Yaskawa INFORM job: apremTRJ3.JBI

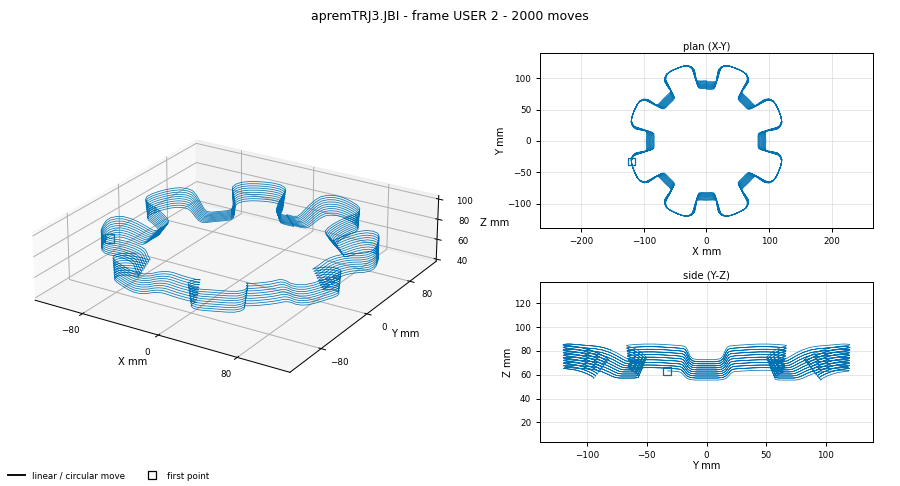
[picture p0: tool path of apremTRJ3.JBI in frame USER 2, 2000 of 2000 moves have a stored position in this frame; points joined in program order, loops and branches not executed]
/JOB
//NAME apremTRJ3
//POS
///NPOS 2000,0,0,0,0,0
///USER 2
///TOOL 1
///POSTYPE USER
///RECTAN
///RCONF 1,0,0,0,0,0,0,0,0,0,0,0,0,0,0,0,0,0,0,0,0,0,0,0
C00000=-119.725,-32.765,63.277,179.9256,-2.1058,0.0000
C00001=-118.418,-27.296,62.983,178.3163,-3.5512,0.0000
C00002=-115.167,-23.366,62.624,174.4376,-3.8430,0.0000
C00003=-110.519,-21.436,61.948,173.6854,-2.2369,0.0000
C00004=-105.464,-19.898,60.600,176.0753,-1.2711,0.0000
C00005=-100.994,-18.424,58.871,-179.3385,0.2539,0.0000
C00006=-97.711,-16.719,57.219,-170.3032,5.9788,0.0000
C00007=-95.932,-14.022,56.034,-167.2384,32.2356,0.0000
C00008=-95.724,-9.298,55.566,179.0443,38.8550,0.0000
C00009=-96.014,-4.602,55.545,177.5469,39.0995,0.0000
C00010=-96.126,0.000,55.559,-179.9998,39.1276,0.0000
C00011=-96.015,4.602,55.545,-177.5472,39.0996,0.0000
C00012=-95.724,9.298,55.566,-179.0464,38.8547,0.0000
C00013=-95.932,14.023,56.035,167.2390,32.2361,0.0000
C00014=-97.711,16.719,57.219,170.3032,5.9788,0.0000
C00015=-100.994,18.424,58.871,179.3385,0.2539,0.0000
C00016=-105.464,19.898,60.600,-176.0753,-1.2711,0.0000
C00017=-110.519,21.436,61.948,-173.6854,-2.2369,0.0000
C00018=-115.167,23.366,62.624,-174.4376,-3.8430,0.0000
C00019=-118.418,27.296,62.983,-178.3163,-3.5512,0.0000
C00020=-119.725,32.765,63.277,-179.9256,-2.1058,0.0000
C00021=-118.751,38.770,63.576,179.9642,-0.1157,0.0000
C00022=-116.678,44.821,63.773,179.9946,-0.0143,0.0000
C00023=-114.197,50.811,63.773,179.9937,-0.0139,0.0000
C00024=-111.384,56.555,63.576,179.9435,-0.1071,0.0000
C00025=-107.827,61.490,63.277,178.4580,-1.4368,0.0000
C00026=-103.035,64.433,62.983,176.3000,-1.3231,0.0000
C00027=-97.958,64.913,62.624,173.3627,1.2239,0.0000
C00028=-93.306,62.991,61.948,173.9567,2.8983,0.0000
C00029=-88.644,60.504,60.600,176.3265,1.8799,0.0000
C00030=-84.442,58.386,58.871,-179.3527,-0.2883,0.0000
C00031=-80.914,57.270,57.219,-168.9722,-2.6779,0.0000
C00032=-77.750,57.919,56.034,-148.7818,15.9473,0.0000
C00033=-74.261,61.112,55.566,-150.8450,30.1755,0.0000
C00034=-71.147,64.638,55.545,-151.4385,31.1712,0.0000
C00035=-67.972,67.972,55.559,-150.0917,29.9081,0.0000
C00036=-64.639,71.146,55.545,-148.8289,28.5617,0.0000
C00037=-61.112,74.261,55.566,-149.8258,29.1559,0.0000
C00038=-57.919,77.750,56.035,-164.0518,31.2182,0.0000
C00039=-57.270,80.914,57.219,177.3221,11.0278,0.0000
C00040=-58.386,84.442,58.871,179.7117,0.6473,0.0000
C00041=-60.504,88.644,60.600,-178.1201,-3.6735,0.0000
C00042=-62.991,93.306,61.948,-177.1017,-6.0433,0.0000
C00043=-64.913,97.958,62.624,-178.7761,-6.6373,0.0000
C00044=-64.433,103.035,62.983,178.6769,-3.7000,0.0000
C00045=-61.490,107.827,63.277,178.5632,-1.5420,0.0000
C00046=-56.555,111.384,63.576,179.8929,-0.0565,0.0000
C00047=-50.811,114.197,63.773,179.9861,-0.0063,0.0000
C00048=-44.821,116.678,63.773,179.9857,-0.0054,0.0000
C00049=-38.770,118.751,63.576,179.8843,-0.0358,0.0000
C00050=-32.765,119.725,63.277,177.8942,0.0744,0.0000
C00051=-27.296,118.418,62.983,176.4488,1.6837,0.0000
C00052=-23.366,115.167,62.624,176.1570,5.5624,0.0000
C00053=-21.436,110.519,61.948,177.7631,6.3146,0.0000
C00054=-19.898,105.464,60.600,178.7289,3.9247,0.0000
C00055=-18.424,100.994,58.871,-179.7461,-0.6615,0.0000
C00056=-16.719,97.711,57.219,-174.0212,-9.6968,0.0000
C00057=-14.023,95.932,56.035,-147.7639,-12.7610,0.0000
C00058=-9.298,95.724,55.566,-141.1453,0.9536,0.0000
C00059=-4.602,96.015,55.545,-140.9004,2.4528,0.0000
C00060=0.000,96.126,55.559,-140.8724,0.0002,0.0000
C00061=0.000,94.736,57.264,-140.7733,0.0001,0.0000
C00062=4.475,94.629,57.250,-140.8009,-2.4427,0.0000
C00063=9.084,94.351,57.271,-141.0650,-0.7004,0.0000
C00064=13.760,94.602,57.767,-148.3519,13.4830,0.0000
C00065=16.395,96.491,59.021,-174.9739,8.8071,0.0000
C00066=18.049,99.951,60.772,-179.9988,0.0034,0.0000
C00067=19.486,104.658,62.604,178.6708,-4.3590,0.0000
C00068=20.989,109.986,64.035,177.7869,-6.6807,0.0000
C00069=22.877,114.901,64.752,176.1277,-5.9675,0.0000
C00070=26.834,118.363,65.133,176.2739,-1.8689,0.0000
C00071=32.398,119.792,65.445,177.8036,-0.1013,0.0000
C00072=38.538,118.828,65.762,179.8764,0.0380,0.0000
C00073=44.742,116.708,65.972,179.9849,0.0057,0.0000
C00074=50.888,114.162,65.972,179.9853,0.0067,0.0000
C00075=56.774,111.274,65.762,179.8857,0.0605,0.0000
C00076=61.797,107.615,65.445,178.5181,1.6250,0.0000
C00077=64.721,102.670,65.133,178.6837,3.9541,0.0000
C00078=65.071,97.424,64.752,-178.5077,6.9431,0.0000
C00079=62.931,92.614,64.035,-176.8235,6.2858,0.0000
C00080=60.226,87.783,62.604,-177.8528,4.0217,0.0000
C00081=57.914,83.439,60.772,179.9985,-0.0033,0.0000
C00082=56.637,79.823,59.021,177.2881,-9.7451,0.0000
C00083=57.164,76.624,57.767,-165.0885,-31.1896,0.0000
C00084=60.292,73.139,57.271,-149.8896,-29.3635,0.0000
C00085=63.749,70.077,57.250,-148.7486,-28.6574,0.0000
C00086=66.989,66.989,57.264,-150.0043,-29.9958,0.0000
C00087=70.077,63.749,57.250,-151.3424,-31.2513,0.0000
C00088=73.140,60.292,57.271,-150.6355,-30.1090,0.0000
C00089=76.624,57.164,57.767,-148.8104,-14.9124,0.0000
C00090=79.823,56.637,59.021,-170.2549,2.7119,0.0000
C00091=83.439,57.914,60.772,-179.9967,0.0015,0.0000
C00092=87.783,60.226,62.604,175.9783,-2.1472,0.0000
C00093=92.614,62.931,64.035,173.7142,-3.1765,0.0000
C00094=97.424,65.071,64.752,173.0569,-1.4923,0.0000
C00095=102.670,64.721,65.133,176.0459,1.3163,0.0000
C00096=107.615,61.797,65.445,178.3750,1.4819,0.0000
C00097=111.274,56.774,65.762,179.9395,0.1143,0.0000
C00098=114.162,50.888,65.972,179.9933,0.0147,0.0000
C00099=116.708,44.742,65.972,179.9943,0.0151,0.0000
C00100=118.828,38.538,65.762,179.9620,0.1236,0.0000
C00101=119.792,32.398,65.445,-179.8987,2.1964,0.0000
C00102=118.363,26.834,65.133,-178.1311,3.7261,0.0000
C00103=114.901,22.877,64.752,-174.0325,3.8723,0.0000
C00104=109.986,20.989,64.035,-173.3193,2.2131,0.0000
C00105=104.658,19.486,62.604,-175.6410,1.3292,0.0000
C00106=99.951,18.049,60.772,179.9966,-0.0012,0.0000
C00107=96.491,16.395,59.021,171.1929,-5.0261,0.0000
C00108=94.602,13.760,57.767,166.5170,-31.6481,0.0000
C00109=94.351,9.084,57.271,-179.2996,-38.9350,0.0000
C00110=94.629,4.475,57.250,-177.5573,-39.1991,0.0000
C00111=94.736,0.000,57.264,179.9999,-39.2267,0.0000
C00112=94.629,-4.475,57.250,177.5575,-39.1991,0.0000
C00113=94.351,-9.084,57.271,179.3018,-38.9347,0.0000
C00114=94.602,-13.760,57.767,-166.5176,-31.6486,0.0000
C00115=96.491,-16.395,59.021,-171.1929,-5.0261,0.0000
C00116=99.951,-18.049,60.772,-179.9966,-0.0012,0.0000
C00117=104.658,-19.486,62.604,175.6410,1.3292,0.0000
C00118=109.986,-20.989,64.035,173.3193,2.2131,0.0000
C00119=114.901,-22.877,64.752,174.0325,3.8723,0.0000
C00120=118.363,-26.834,65.133,178.1311,3.7261,0.0000
C00121=119.792,-32.398,65.445,179.8987,2.1964,0.0000
C00122=118.828,-38.538,65.762,-179.9620,0.1236,0.0000
C00123=116.708,-44.742,65.972,-179.9943,0.0151,0.0000
C00124=114.162,-50.888,65.972,-179.9933,0.0147,0.0000
C00125=111.274,-56.774,65.762,-179.9395,0.1143,0.0000
C00126=107.615,-61.797,65.445,-178.3750,1.4819,0.0000
C00127=102.670,-64.721,65.133,-176.0459,1.3163,0.0000
C00128=97.424,-65.071,64.752,-173.0569,-1.4923,0.0000
C00129=92.614,-62.931,64.035,-173.7142,-3.1765,0.0000
C00130=87.783,-60.226,62.604,-175.9783,-2.1472,0.0000
C00131=83.439,-57.914,60.772,179.9967,0.0015,0.0000
C00132=79.823,-56.637,59.021,170.2549,2.7119,0.0000
C00133=76.624,-57.164,57.767,148.8104,-14.9115,0.0000
C00134=73.139,-60.292,57.271,150.6365,-30.1104,0.0000
C00135=70.077,-63.749,57.250,151.3426,-31.2514,0.0000
C00136=66.989,-66.989,57.264,150.0042,-29.9957,0.0000
C00137=63.749,-70.077,57.250,148.7487,-28.6576,0.0000
C00138=60.292,-73.140,57.271,149.8910,-29.3645,0.0000
C00139=57.164,-76.624,57.767,165.0876,-31.1896,0.0000
C00140=56.637,-79.823,59.021,-177.2881,-9.7451,0.0000
C00141=57.914,-83.439,60.772,-179.9985,-0.0033,0.0000
C00142=60.226,-87.783,62.604,177.8528,4.0217,0.0000
C00143=62.931,-92.614,64.035,176.8235,6.2858,0.0000
C00144=65.071,-97.424,64.752,178.5077,6.9431,0.0000
C00145=64.721,-102.670,65.133,-178.6837,3.9541,0.0000
C00146=61.797,-107.615,65.445,-178.5181,1.6250,0.0000
C00147=56.774,-111.274,65.762,-179.8857,0.0605,0.0000
C00148=50.888,-114.162,65.972,-179.9853,0.0067,0.0000
C00149=44.742,-116.708,65.972,-179.9849,0.0057,0.0000
C00150=38.538,-118.828,65.762,-179.8764,0.0380,0.0000
C00151=32.398,-119.792,65.445,-177.8036,-0.1013,0.0000
C00152=26.834,-118.363,65.133,-176.2739,-1.8689,0.0000
C00153=22.877,-114.901,64.752,-176.1277,-5.9675,0.0000
C00154=20.989,-109.986,64.035,-177.7869,-6.6807,0.0000
C00155=19.486,-104.658,62.604,-178.6708,-4.3590,0.0000
C00156=18.049,-99.951,60.772,179.9988,0.0034,0.0000
C00157=16.395,-96.491,59.021,174.9739,8.8071,0.0000
C00158=13.760,-94.602,57.767,148.3519,13.4830,0.0000
C00159=9.084,-94.351,57.271,141.0650,-0.7004,0.0000
C00160=4.475,-94.629,57.250,140.8009,-2.4427,0.0000
C00161=0.000,-94.736,57.264,140.7733,0.0001,0.0000
C00162=0.000,-94.736,57.264,140.7733,0.0001,0.0000
C00163=-4.475,-94.629,57.250,140.8009,2.4425,0.0000
C00164=-9.084,-94.351,57.271,141.0653,0.6982,0.0000
C00165=-13.760,-94.602,57.767,148.3514,-13.4824,0.0000
C00166=-16.395,-96.491,59.021,174.9739,-8.8071,0.0000
C00167=-18.049,-99.951,60.772,179.9988,-0.0034,0.0000
C00168=-19.486,-104.658,62.604,-178.6708,4.3590,0.0000
C00169=-20.989,-109.986,64.035,-177.7869,6.6807,0.0000
C00170=-22.877,-114.901,64.752,-176.1277,5.9675,0.0000
C00171=-26.834,-118.363,65.133,-176.2739,1.8689,0.0000
C00172=-32.398,-119.792,65.445,-177.8036,0.1013,0.0000
C00173=-38.538,-118.828,65.762,-179.8764,-0.0380,0.0000
C00174=-44.742,-116.708,65.972,-179.9849,-0.0057,0.0000
C00175=-50.888,-114.162,65.972,-179.9853,-0.0067,0.0000
C00176=-56.774,-111.274,65.762,-179.8857,-0.0605,0.0000
C00177=-61.797,-107.615,65.445,-178.5181,-1.6250,0.0000
C00178=-64.721,-102.670,65.133,-178.6837,-3.9541,0.0000
C00179=-65.071,-97.424,64.752,178.5077,-6.9431,0.0000
C00180=-62.931,-92.614,64.035,176.8235,-6.2858,0.0000
C00181=-60.226,-87.783,62.604,177.8528,-4.0217,0.0000
C00182=-57.914,-83.439,60.772,-179.9985,0.0033,0.0000
C00183=-56.637,-79.823,59.021,-177.2881,9.7451,0.0000
C00184=-57.164,-76.624,57.767,165.0885,31.1896,0.0000
C00185=-60.292,-73.139,57.271,149.8896,29.3635,0.0000
C00186=-63.749,-70.077,57.250,148.7486,28.6574,0.0000
C00187=-66.989,-66.989,57.264,150.0043,29.9958,0.0000
C00188=-70.077,-63.749,57.250,151.3424,31.2513,0.0000
C00189=-73.140,-60.292,57.271,150.6355,30.1090,0.0000
C00190=-76.624,-57.164,57.767,148.8104,14.9124,0.0000
C00191=-79.823,-56.637,59.021,170.2549,-2.7119,0.0000
C00192=-83.439,-57.914,60.772,179.9967,-0.0015,0.0000
C00193=-87.783,-60.226,62.604,-175.9783,2.1472,0.0000
C00194=-92.614,-62.931,64.035,-173.7142,3.1765,0.0000
C00195=-97.424,-65.071,64.752,-173.0569,1.4923,0.0000
C00196=-102.670,-64.721,65.133,-176.0459,-1.3163,0.0000
C00197=-107.615,-61.797,65.445,-178.3750,-1.4819,0.0000
C00198=-111.274,-56.774,65.762,-179.9395,-0.1143,0.0000
C00199=-114.162,-50.888,65.972,-179.9933,-0.0147,0.0000
C00200=-116.708,-44.742,65.972,-179.9943,-0.0151,0.0000
C00201=-118.828,-38.538,65.762,-179.9620,-0.1236,0.0000
C00202=-119.792,-32.398,65.445,179.8987,-2.1964,0.0000
C00203=-118.363,-26.834,65.133,178.1311,-3.7261,0.0000
C00204=-114.901,-22.877,64.752,174.0325,-3.8723,0.0000
C00205=-109.986,-20.989,64.035,173.3193,-2.2131,0.0000
C00206=-104.658,-19.486,62.604,175.6410,-1.3292,0.0000
C00207=-99.951,-18.049,60.772,-179.9966,0.0012,0.0000
C00208=-96.491,-16.395,59.021,-171.1929,5.0261,0.0000
C00209=-94.602,-13.760,57.767,-166.5170,31.6481,0.0000
C00210=-94.351,-9.084,57.271,179.2996,38.9350,0.0000
C00211=-94.629,-4.475,57.250,177.5573,39.1991,0.0000
C00212=-94.736,0.000,57.264,-179.9999,39.2267,0.0000
C00213=-94.629,4.475,57.250,-177.5575,39.1991,0.0000
C00214=-94.351,9.084,57.271,-179.3018,38.9347,0.0000
C00215=-94.602,13.760,57.767,166.5176,31.6486,0.0000
C00216=-96.491,16.395,59.021,171.1929,5.0261,0.0000
C00217=-99.951,18.049,60.772,179.9966,0.0012,0.0000
C00218=-104.658,19.486,62.604,-175.6410,-1.3292,0.0000
C00219=-109.986,20.989,64.035,-173.3193,-2.2131,0.0000
C00220=-114.901,22.877,64.752,-174.0325,-3.8723,0.0000
C00221=-118.363,26.834,65.133,-178.1311,-3.7261,0.0000
C00222=-119.792,32.398,65.445,-179.8987,-2.1964,0.0000
C00223=-118.828,38.538,65.762,179.9620,-0.1236,0.0000
C00224=-116.708,44.742,65.972,179.9943,-0.0151,0.0000
C00225=-114.162,50.888,65.972,179.9933,-0.0147,0.0000
C00226=-111.274,56.774,65.762,179.9395,-0.1143,0.0000
C00227=-107.615,61.797,65.445,178.3750,-1.4819,0.0000
C00228=-102.670,64.721,65.133,176.0459,-1.3163,0.0000
C00229=-97.424,65.071,64.752,173.0569,1.4923,0.0000
C00230=-92.614,62.931,64.035,173.7142,3.1765,0.0000
C00231=-87.783,60.226,62.604,175.9783,2.1472,0.0000
C00232=-83.439,57.914,60.772,-179.9967,-0.0015,0.0000
C00233=-79.823,56.637,59.021,-170.2549,-2.7119,0.0000
C00234=-76.624,57.164,57.767,-148.8104,14.9115,0.0000
C00235=-73.139,60.292,57.271,-150.6365,30.1104,0.0000
C00236=-70.077,63.749,57.250,-151.3426,31.2514,0.0000
C00237=-66.989,66.989,57.264,-150.0042,29.9957,0.0000
C00238=-63.749,70.077,57.250,-148.7487,28.6576,0.0000
C00239=-60.292,73.140,57.271,-149.8910,29.3645,0.0000
C00240=-57.164,76.624,57.767,-165.0876,31.1896,0.0000
C00241=-56.637,79.823,59.021,177.2881,9.7451,0.0000
C00242=-57.914,83.439,60.772,179.9985,0.0033,0.0000
C00243=-60.226,87.783,62.604,-177.8528,-4.0217,0.0000
C00244=-62.931,92.614,64.035,-176.8235,-6.2858,0.0000
C00245=-65.071,97.424,64.752,-178.5077,-6.9431,0.0000
C00246=-64.721,102.670,65.133,178.6837,-3.9541,0.0000
C00247=-61.797,107.615,65.445,178.5181,-1.6250,0.0000
C00248=-56.774,111.274,65.762,179.8857,-0.0605,0.0000
C00249=-50.888,114.162,65.972,179.9853,-0.0067,0.0000
C00250=-44.742,116.708,65.972,179.9849,-0.0057,0.0000
C00251=-38.538,118.828,65.762,179.8764,-0.0380,0.0000
C00252=-32.398,119.792,65.445,177.8036,0.1013,0.0000
C00253=-26.834,118.363,65.133,176.2739,1.8689,0.0000
C00254=-22.877,114.901,64.752,176.1277,5.9675,0.0000
C00255=-20.989,109.986,64.035,177.7869,6.6807,0.0000
C00256=-19.486,104.658,62.604,178.6708,4.3590,0.0000
C00257=-18.049,99.951,60.772,-179.9988,-0.0034,0.0000
C00258=-16.395,96.491,59.021,-174.9739,-8.8071,0.0000
C00259=-13.760,94.602,57.767,-148.3514,-13.4824,0.0000
C00260=-9.084,94.351,57.271,-141.0653,0.6982,0.0000
C00261=-4.475,94.629,57.250,-140.8009,2.4425,0.0000
C00262=0.000,94.736,57.264,-140.7733,0.0001,0.0000
C00263=0.000,93.344,58.968,-140.7215,0.0000,0.0000
C00264=4.348,93.242,58.953,-140.7485,-2.4271,0.0000
C00265=8.870,92.975,58.975,-141.0344,-0.4357,0.0000
C00266=13.498,93.270,59.499,-149.0201,14.1329,0.0000
C00267=16.071,95.271,60.823,-175.8165,7.9019,0.0000
C00268=17.674,98.909,62.673,179.7950,-0.6064,0.0000
C00269=19.074,103.853,64.610,178.6348,-4.7423,0.0000
C00270=20.544,109.456,66.124,177.8284,-6.9903,0.0000
C00271=22.391,114.637,66.882,176.1347,-6.3202,0.0000
C00272=26.375,118.308,67.284,176.1293,-2.0440,0.0000
C00273=32.034,119.858,67.614,177.7255,-0.1282,0.0000
C00274=38.307,118.904,67.949,179.8694,0.0400,0.0000
C00275=44.664,116.738,68.170,179.9841,0.0060,0.0000
C00276=50.965,114.128,68.170,179.9845,0.0070,0.0000
C00277=56.991,111.165,67.949,179.8794,0.0641,0.0000
C00278=62.101,107.404,67.614,178.4818,1.6994,0.0000
C00279=65.006,102.306,67.284,178.7050,4.1797,0.0000
C00280=65.228,96.893,66.882,-178.2506,7.1867,0.0000
C00281=62.871,91.924,66.124,-176.5728,6.4761,0.0000
C00282=59.948,86.923,64.610,-177.6059,4.3183,0.0000
C00283=57.442,82.437,62.673,-179.7162,0.5738,0.0000
C00284=56.002,78.731,60.823,177.3422,-8.5232,0.0000
C00285=56.408,75.496,59.499,-166.1532,-31.0723,0.0000
C00286=59.471,72.016,58.975,-150.0031,-29.5326,0.0000
C00287=62.858,69.007,58.953,-148.7116,-28.7135,0.0000
C00288=66.004,66.004,58.968,-149.9585,-30.0416,0.0000
C00289=69.006,62.858,58.953,-151.2864,-31.2884,0.0000
C00290=72.016,59.471,58.975,-150.4665,-29.9954,0.0000
C00291=75.496,56.408,59.499,-148.9276,-13.8477,0.0000
C00292=78.731,56.002,60.823,-171.4768,2.6578,0.0000
C00293=82.437,57.442,62.673,179.4262,-0.2838,0.0000
C00294=86.923,59.948,64.610,175.6817,-2.3941,0.0000
C00295=91.924,62.871,66.124,173.5239,-3.4272,0.0000
C00296=96.893,65.228,66.882,172.8133,-1.7494,0.0000
C00297=102.306,65.006,67.284,175.8203,1.2950,0.0000
C00298=107.404,62.101,67.614,178.3006,1.5182,0.0000
C00299=111.165,56.991,67.949,179.9359,0.1206,0.0000
C00300=114.128,50.965,68.170,179.9930,0.0155,0.0000
C00301=116.738,44.664,68.170,179.9940,0.0159,0.0000
C00302=118.904,38.307,67.949,179.9600,0.1306,0.0000
C00303=119.858,32.034,67.614,-179.8718,2.2745,0.0000
C00304=118.308,26.375,67.284,-177.9560,3.8707,0.0000
C00305=114.637,22.391,66.882,-173.6798,3.8653,0.0000
C00306=109.456,20.544,66.124,-173.0097,2.1716,0.0000
C00307=103.853,19.074,64.610,-175.2577,1.3652,0.0000
C00308=98.909,17.674,62.673,-179.3936,0.2050,0.0000
C00309=95.271,16.071,60.823,172.0981,-4.1835,0.0000
C00310=93.270,13.498,59.499,165.8671,-30.9799,0.0000
C00311=92.975,8.870,58.975,-179.5643,-38.9656,0.0000
C00312=93.242,4.348,58.953,-177.5729,-39.2515,0.0000
C00313=93.344,0.000,58.968,180.0000,-39.2785,0.0000
C00314=93.242,-4.348,58.953,177.5731,-39.2515,0.0000
C00315=92.976,-8.870,58.975,179.5666,-38.9653,0.0000
C00316=93.271,-13.498,59.499,-165.8676,-30.9804,0.0000
C00317=95.271,-16.071,60.823,-172.0981,-4.1835,0.0000
C00318=98.909,-17.674,62.673,179.3936,0.2050,0.0000
C00319=103.853,-19.074,64.610,175.2577,1.3652,0.0000
C00320=109.456,-20.544,66.124,173.0097,2.1716,0.0000
C00321=114.637,-22.391,66.882,173.6798,3.8653,0.0000
C00322=118.308,-26.375,67.284,177.9560,3.8707,0.0000
C00323=119.858,-32.034,67.614,179.8718,2.2745,0.0000
C00324=118.904,-38.307,67.949,-179.9600,0.1306,0.0000
C00325=116.738,-44.664,68.170,-179.9940,0.0159,0.0000
C00326=114.128,-50.965,68.170,-179.9930,0.0155,0.0000
C00327=111.165,-56.991,67.949,-179.9359,0.1206,0.0000
C00328=107.404,-62.101,67.614,-178.3006,1.5182,0.0000
C00329=102.306,-65.006,67.284,-175.8203,1.2950,0.0000
C00330=96.893,-65.228,66.882,-172.8133,-1.7494,0.0000
C00331=91.924,-62.871,66.124,-173.5239,-3.4272,0.0000
C00332=86.923,-59.948,64.610,-175.6817,-2.3941,0.0000
C00333=82.437,-57.442,62.673,-179.4262,-0.2838,0.0000
C00334=78.731,-56.002,60.823,171.4768,2.6578,0.0000
C00335=75.496,-56.408,59.499,148.9277,-13.8468,0.0000
C00336=72.016,-59.471,58.975,150.4674,-29.9969,0.0000
C00337=69.007,-62.858,58.953,151.2865,-31.2884,0.0000
C00338=66.004,-66.004,58.968,149.9584,-30.0415,0.0000
C00339=62.858,-69.006,58.953,148.7116,-28.7136,0.0000
C00340=59.471,-72.016,58.975,150.0046,-29.5335,0.0000
C00341=56.408,-75.496,59.499,166.1523,-31.0724,0.0000
C00342=56.002,-78.731,60.823,-177.3422,-8.5232,0.0000
C00343=57.442,-82.437,62.673,179.7162,0.5738,0.0000
C00344=59.948,-86.923,64.610,177.6059,4.3183,0.0000
C00345=62.871,-91.924,66.124,176.5728,6.4761,0.0000
C00346=65.228,-96.893,66.882,178.2506,7.1867,0.0000
C00347=65.006,-102.306,67.284,-178.7050,4.1797,0.0000
C00348=62.101,-107.404,67.614,-178.4818,1.6994,0.0000
C00349=56.991,-111.165,67.949,-179.8794,0.0641,0.0000
C00350=50.965,-114.128,68.170,-179.9845,0.0070,0.0000
C00351=44.664,-116.738,68.170,-179.9841,0.0060,0.0000
C00352=38.307,-118.904,67.949,-179.8694,0.0400,0.0000
C00353=32.034,-119.858,67.614,-177.7255,-0.1282,0.0000
C00354=26.375,-118.308,67.284,-176.1293,-2.0440,0.0000
C00355=22.391,-114.637,66.882,-176.1347,-6.3202,0.0000
C00356=20.544,-109.456,66.124,-177.8284,-6.9903,0.0000
C00357=19.074,-103.853,64.610,-178.6348,-4.7423,0.0000
C00358=17.674,-98.909,62.673,-179.7950,-0.6064,0.0000
C00359=16.071,-95.271,60.823,175.8165,7.9019,0.0000
C00360=13.498,-93.270,59.499,149.0201,14.1329,0.0000
C00361=8.870,-92.975,58.975,141.0344,-0.4357,0.0000
C00362=4.348,-93.242,58.953,140.7485,-2.4271,0.0000
C00363=0.000,-93.344,58.968,140.7215,0.0000,0.0000
C00364=0.000,-93.344,58.968,140.7215,0.0000,0.0000
C00365=-4.348,-93.242,58.953,140.7485,2.4269,0.0000
C00366=-8.870,-92.976,58.975,141.0347,0.4334,0.0000
C00367=-13.498,-93.271,59.499,149.0196,-14.1324,0.0000
C00368=-16.071,-95.271,60.823,175.8165,-7.9019,0.0000
C00369=-17.674,-98.909,62.673,-179.7950,0.6064,0.0000
C00370=-19.074,-103.853,64.610,-178.6348,4.7423,0.0000
C00371=-20.544,-109.456,66.124,-177.8284,6.9903,0.0000
C00372=-22.391,-114.637,66.882,-176.1347,6.3202,0.0000
C00373=-26.375,-118.308,67.284,-176.1293,2.0440,0.0000
C00374=-32.034,-119.858,67.614,-177.7255,0.1282,0.0000
C00375=-38.307,-118.904,67.949,-179.8694,-0.0400,0.0000
C00376=-44.664,-116.738,68.170,-179.9841,-0.0060,0.0000
C00377=-50.965,-114.128,68.170,-179.9845,-0.0070,0.0000
C00378=-56.991,-111.165,67.949,-179.8794,-0.0641,0.0000
C00379=-62.101,-107.404,67.614,-178.4818,-1.6994,0.0000
C00380=-65.006,-102.306,67.284,-178.7050,-4.1797,0.0000
C00381=-65.228,-96.893,66.882,178.2506,-7.1867,0.0000
C00382=-62.871,-91.924,66.124,176.5728,-6.4761,0.0000
C00383=-59.948,-86.923,64.610,177.6059,-4.3183,0.0000
C00384=-57.442,-82.437,62.673,179.7162,-0.5738,0.0000
C00385=-56.002,-78.731,60.823,-177.3422,8.5232,0.0000
C00386=-56.408,-75.496,59.499,166.1532,31.0723,0.0000
C00387=-59.471,-72.016,58.975,150.0031,29.5326,0.0000
C00388=-62.858,-69.007,58.953,148.7116,28.7135,0.0000
C00389=-66.004,-66.004,58.968,149.9585,30.0416,0.0000
C00390=-69.006,-62.858,58.953,151.2864,31.2884,0.0000
C00391=-72.016,-59.471,58.975,150.4665,29.9954,0.0000
C00392=-75.496,-56.408,59.499,148.9276,13.8477,0.0000
C00393=-78.731,-56.002,60.823,171.4768,-2.6578,0.0000
C00394=-82.437,-57.442,62.673,-179.4262,0.2838,0.0000
C00395=-86.923,-59.948,64.610,-175.6817,2.3941,0.0000
C00396=-91.924,-62.871,66.124,-173.5239,3.4272,0.0000
C00397=-96.893,-65.228,66.882,-172.8133,1.7494,0.0000
C00398=-102.306,-65.006,67.284,-175.8203,-1.2950,0.0000
C00399=-107.404,-62.101,67.614,-178.3006,-1.5182,0.0000
C00400=-111.165,-56.991,67.949,-179.9359,-0.1206,0.0000
C00401=-114.128,-50.965,68.170,-179.9930,-0.0155,0.0000
C00402=-116.738,-44.664,68.170,-179.9940,-0.0159,0.0000
C00403=-118.904,-38.307,67.949,-179.9600,-0.1306,0.0000
C00404=-119.858,-32.034,67.614,179.8718,-2.2745,0.0000
C00405=-118.308,-26.375,67.284,177.9560,-3.8707,0.0000
C00406=-114.637,-22.391,66.882,173.6798,-3.8653,0.0000
C00407=-109.456,-20.544,66.124,173.0097,-2.1716,0.0000
C00408=-103.853,-19.074,64.610,175.2577,-1.3652,0.0000
C00409=-98.909,-17.674,62.673,179.3936,-0.2050,0.0000
C00410=-95.271,-16.071,60.823,-172.0981,4.1835,0.0000
C00411=-93.270,-13.498,59.499,-165.8671,30.9799,0.0000
C00412=-92.975,-8.870,58.975,179.5643,38.9656,0.0000
C00413=-93.242,-4.348,58.953,177.5729,39.2515,0.0000
C00414=-93.344,0.000,58.968,-180.0000,39.2785,0.0000
C00415=-93.242,4.348,58.953,-177.5731,39.2515,0.0000
C00416=-92.976,8.870,58.975,-179.5666,38.9653,0.0000
C00417=-93.271,13.498,59.499,165.8676,30.9804,0.0000
C00418=-95.271,16.071,60.823,172.0981,4.1835,0.0000
C00419=-98.909,17.674,62.673,-179.3936,-0.2050,0.0000
C00420=-103.853,19.074,64.610,-175.2577,-1.3652,0.0000
C00421=-109.456,20.544,66.124,-173.0097,-2.1716,0.0000
C00422=-114.637,22.391,66.882,-173.6798,-3.8653,0.0000
C00423=-118.308,26.375,67.284,-177.9560,-3.8707,0.0000
C00424=-119.858,32.034,67.614,-179.8718,-2.2745,0.0000
C00425=-118.904,38.307,67.949,179.9600,-0.1306,0.0000
C00426=-116.738,44.664,68.170,179.9940,-0.0159,0.0000
C00427=-114.128,50.965,68.170,179.9930,-0.0155,0.0000
C00428=-111.165,56.991,67.949,179.9359,-0.1206,0.0000
C00429=-107.404,62.101,67.614,178.3006,-1.5182,0.0000
C00430=-102.306,65.006,67.284,175.8203,-1.2950,0.0000
C00431=-96.893,65.228,66.882,172.8133,1.7494,0.0000
C00432=-91.924,62.871,66.124,173.5239,3.4272,0.0000
C00433=-86.923,59.948,64.610,175.6817,2.3941,0.0000
C00434=-82.437,57.442,62.673,179.4262,0.2838,0.0000
C00435=-78.731,56.002,60.823,-171.4768,-2.6578,0.0000
C00436=-75.496,56.408,59.499,-148.9277,13.8468,0.0000
C00437=-72.016,59.471,58.975,-150.4674,29.9969,0.0000
C00438=-69.007,62.858,58.953,-151.2865,31.2884,0.0000
C00439=-66.004,66.004,58.968,-149.9584,30.0415,0.0000
C00440=-62.858,69.006,58.953,-148.7116,28.7136,0.0000
C00441=-59.471,72.016,58.975,-150.0046,29.5335,0.0000
C00442=-56.408,75.496,59.499,-166.1523,31.0724,0.0000
C00443=-56.002,78.731,60.823,177.3422,8.5232,0.0000
C00444=-57.442,82.437,62.673,-179.7162,-0.5738,0.0000
C00445=-59.948,86.923,64.610,-177.6059,-4.3183,0.0000
C00446=-62.871,91.924,66.124,-176.5728,-6.4761,0.0000
C00447=-65.228,96.893,66.882,-178.2506,-7.1867,0.0000
C00448=-65.006,102.306,67.284,178.7050,-4.1797,0.0000
C00449=-62.101,107.404,67.614,178.4818,-1.6994,0.0000
C00450=-56.991,111.165,67.949,179.8794,-0.0641,0.0000
C00451=-50.965,114.128,68.170,179.9845,-0.0070,0.0000
C00452=-44.664,116.738,68.170,179.9841,-0.0060,0.0000
C00453=-38.307,118.904,67.949,179.8694,-0.0400,0.0000
C00454=-32.034,119.858,67.614,177.7255,0.1282,0.0000
C00455=-26.375,118.308,67.284,176.1293,2.0440,0.0000
C00456=-22.391,114.637,66.882,176.1347,6.3202,0.0000
C00457=-20.544,109.456,66.124,177.8284,6.9903,0.0000
C00458=-19.074,103.853,64.610,178.6348,4.7423,0.0000
C00459=-17.674,98.909,62.673,179.7950,0.6064,0.0000
C00460=-16.071,95.271,60.823,-175.8165,-7.9019,0.0000
C00461=-13.498,93.271,59.499,-149.0196,-14.1324,0.0000
C00462=-8.870,92.976,58.975,-141.0347,0.4334,0.0000
C00463=-4.348,93.242,58.953,-140.7485,2.4269,0.0000
C00464=0.000,93.344,58.968,-140.7215,0.0000,0.0000
C00465=0.000,91.951,60.671,-140.7165,-0.0000,0.0000
C00466=4.221,91.854,60.655,-140.7430,-2.4062,0.0000
C00467=8.656,91.600,60.679,-141.0531,-0.1630,0.0000
C00468=13.235,91.938,61.230,-149.7643,14.7062,0.0000
C00469=15.748,94.051,62.625,-176.5558,6.9972,0.0000
C00470=17.300,97.869,64.575,179.6283,-1.1669,0.0000
C00471=18.664,103.053,66.618,178.6171,-5.0759,0.0000
C00472=20.101,108.929,68.213,177.8838,-7.2452,0.0000
C00473=21.908,114.374,69.012,176.1721,-6.6194,0.0000
C00474=25.920,118.253,69.436,176.0147,-2.2065,0.0000
C00475=31.673,119.924,69.783,177.6602,-0.1548,0.0000
C00476=38.079,118.979,70.135,179.8633,0.0417,0.0000
C00477=44.586,116.768,70.368,179.9835,0.0062,0.0000
C00478=51.040,114.095,70.368,179.9839,0.0073,0.0000
C00479=57.205,111.057,70.135,179.8739,0.0672,0.0000
C00480=62.403,107.195,69.783,178.4545,1.7643,0.0000
C00481=65.289,101.946,69.436,178.7386,4.3750,0.0000
C00482=65.383,96.366,69.012,-178.0100,7.3714,0.0000
C00483=62.811,91.238,68.213,-176.3515,6.6181,0.0000
C00484=59.672,86.067,66.618,-177.3813,4.5670,0.0000
C00485=56.971,81.437,64.575,-179.4376,1.0880,0.0000
C00486=55.369,77.639,62.625,177.4675,-7.3700,0.0000
C00487=55.652,74.369,61.230,-167.2352,-30.8677,0.0000
C00488=58.650,70.891,60.679,-150.1644,-29.6618,0.0000
C00489=61.966,67.935,60.655,-148.7176,-28.7299,0.0000
C00490=65.019,65.019,60.671,-149.9540,-30.0459,0.0000
C00491=67.935,61.966,60.655,-151.2700,-31.2824,0.0000
C00492=70.892,58.650,60.679,-150.3372,-29.8340,0.0000
C00493=74.369,55.652,61.230,-149.1322,-12.7656,0.0000
C00494=77.639,55.369,62.625,-172.6300,2.5325,0.0000
C00495=81.437,56.971,64.575,178.9120,-0.5624,0.0000
C00496=86.067,59.672,66.618,175.4330,-2.6187,0.0000
C00497=91.238,62.811,68.213,173.3819,-3.6485,0.0000
C00498=96.366,65.383,69.012,172.6286,-1.9900,0.0000
C00499=101.946,65.289,69.436,175.6250,1.2614,0.0000
C00500=107.195,62.403,69.783,178.2357,1.5455,0.0000
C00501=111.057,57.205,70.135,179.9328,0.1261,0.0000
C00502=114.095,51.040,70.368,179.9927,0.0161,0.0000
C00503=116.768,44.586,70.368,179.9938,0.0165,0.0000
C00504=118.979,38.079,70.135,179.9583,0.1367,0.0000
C00505=119.924,31.673,69.783,-179.8452,2.3398,0.0000
C00506=118.253,25.920,69.436,-177.7935,3.9853,0.0000
C00507=114.374,21.908,69.012,-173.3806,3.8279,0.0000
C00508=108.929,20.101,68.213,-172.7548,2.1162,0.0000
C00509=103.053,18.664,66.618,-174.9241,1.3829,0.0000
C00510=97.869,17.300,64.575,-178.8331,0.3717,0.0000
C00511=94.051,15.748,62.625,173.0028,-3.4442,0.0000
C00512=91.938,13.235,61.230,165.2938,-30.2357,0.0000
C00513=91.600,8.656,60.679,-179.8370,-38.9469,0.0000
C00514=91.854,4.221,60.655,-177.5938,-39.2570,0.0000
C00515=91.951,0.000,60.671,-180.0000,-39.2835,0.0000
C00516=91.854,-4.220,60.655,177.5939,-39.2571,0.0000
C00517=91.600,-8.656,60.679,179.8394,-38.9465,0.0000
C00518=91.938,-13.235,61.230,-165.2943,-30.2362,0.0000
C00519=94.051,-15.748,62.625,-173.0028,-3.4442,0.0000
C00520=97.869,-17.300,64.575,178.8331,0.3717,0.0000
C00521=103.053,-18.664,66.618,174.9241,1.3829,0.0000
C00522=108.929,-20.101,68.213,172.7548,2.1162,0.0000
C00523=114.374,-21.908,69.012,173.3806,3.8279,0.0000
C00524=118.253,-25.920,69.436,177.7935,3.9853,0.0000
C00525=119.924,-31.673,69.783,179.8452,2.3398,0.0000
C00526=118.979,-38.079,70.135,-179.9583,0.1367,0.0000
C00527=116.768,-44.586,70.368,-179.9938,0.0165,0.0000
C00528=114.095,-51.040,70.368,-179.9927,0.0161,0.0000
C00529=111.057,-57.205,70.135,-179.9328,0.1261,0.0000
C00530=107.195,-62.403,69.783,-178.2357,1.5455,0.0000
C00531=101.946,-65.289,69.436,-175.6250,1.2614,0.0000
C00532=96.366,-65.383,69.012,-172.6286,-1.9900,0.0000
C00533=91.238,-62.811,68.213,-173.3819,-3.6485,0.0000
C00534=86.067,-59.672,66.618,-175.4330,-2.6187,0.0000
C00535=81.437,-56.971,64.575,-178.9120,-0.5624,0.0000
C00536=77.639,-55.369,62.625,172.6300,2.5325,0.0000
C00537=74.369,-55.652,61.230,149.1323,-12.7648,0.0000
C00538=70.891,-58.650,60.679,150.3382,-29.8356,0.0000
C00539=67.935,-61.966,60.655,151.2701,-31.2824,0.0000
C00540=65.019,-65.019,60.671,149.9541,-30.0460,0.0000
C00541=61.966,-67.935,60.655,148.7176,-28.7300,0.0000
C00542=58.650,-70.892,60.679,150.1660,-29.6628,0.0000
C00543=55.652,-74.369,61.230,167.2344,-30.8678,0.0000
C00544=55.369,-77.639,62.625,-177.4675,-7.3700,0.0000
C00545=56.971,-81.437,64.575,179.4376,1.0880,0.0000
C00546=59.672,-86.067,66.618,177.3813,4.5670,0.0000
C00547=62.811,-91.238,68.213,176.3515,6.6181,0.0000
C00548=65.383,-96.366,69.012,178.0100,7.3714,0.0000
C00549=65.289,-101.946,69.436,-178.7386,4.3750,0.0000
C00550=62.403,-107.195,69.783,-178.4545,1.7643,0.0000
C00551=57.205,-111.057,70.135,-179.8739,0.0672,0.0000
C00552=51.040,-114.095,70.368,-179.9839,0.0073,0.0000
C00553=44.586,-116.768,70.368,-179.9835,0.0062,0.0000
C00554=38.079,-118.979,70.135,-179.8633,0.0417,0.0000
C00555=31.673,-119.924,69.783,-177.6602,-0.1548,0.0000
C00556=25.920,-118.253,69.436,-176.0147,-2.2065,0.0000
C00557=21.908,-114.374,69.012,-176.1721,-6.6194,0.0000
C00558=20.101,-108.929,68.213,-177.8838,-7.2452,0.0000
C00559=18.664,-103.053,66.618,-178.6171,-5.0759,0.0000
C00560=17.300,-97.869,64.575,-179.6283,-1.1669,0.0000
C00561=15.748,-94.051,62.625,176.5558,6.9972,0.0000
C00562=13.235,-91.938,61.230,149.7643,14.7062,0.0000
C00563=8.656,-91.600,60.679,141.0531,-0.1630,0.0000
C00564=4.221,-91.854,60.655,140.7430,-2.4062,0.0000
C00565=0.000,-91.951,60.671,140.7165,-0.0000,0.0000
C00566=0.000,-91.951,60.671,140.7165,-0.0000,0.0000
C00567=-4.220,-91.854,60.655,140.7429,2.4061,0.0000
C00568=-8.656,-91.600,60.679,141.0535,0.1606,0.0000
C00569=-13.235,-91.938,61.230,149.7638,-14.7057,0.0000
C00570=-15.748,-94.051,62.625,176.5558,-6.9972,0.0000
C00571=-17.300,-97.869,64.575,-179.6283,1.1669,0.0000
C00572=-18.664,-103.053,66.618,-178.6171,5.0759,0.0000
C00573=-20.101,-108.929,68.213,-177.8838,7.2452,0.0000
C00574=-21.908,-114.374,69.012,-176.1721,6.6194,0.0000
C00575=-25.920,-118.253,69.436,-176.0147,2.2065,0.0000
C00576=-31.673,-119.924,69.783,-177.6602,0.1548,0.0000
C00577=-38.079,-118.979,70.135,-179.8633,-0.0417,0.0000
C00578=-44.586,-116.768,70.368,-179.9835,-0.0062,0.0000
C00579=-51.040,-114.095,70.368,-179.9839,-0.0073,0.0000
C00580=-57.205,-111.057,70.135,-179.8739,-0.0672,0.0000
C00581=-62.403,-107.195,69.783,-178.4545,-1.7643,0.0000
C00582=-65.289,-101.946,69.436,-178.7386,-4.3750,0.0000
C00583=-65.383,-96.366,69.012,178.0100,-7.3714,0.0000
C00584=-62.811,-91.238,68.213,176.3515,-6.6181,0.0000
C00585=-59.672,-86.067,66.618,177.3813,-4.5670,0.0000
C00586=-56.971,-81.437,64.575,179.4376,-1.0880,0.0000
C00587=-55.369,-77.639,62.625,-177.4675,7.3700,0.0000
C00588=-55.652,-74.369,61.230,167.2352,30.8677,0.0000
C00589=-58.650,-70.891,60.679,150.1644,29.6618,0.0000
C00590=-61.966,-67.935,60.655,148.7176,28.7299,0.0000
C00591=-65.019,-65.019,60.671,149.9540,30.0459,0.0000
C00592=-67.935,-61.966,60.655,151.2700,31.2824,0.0000
C00593=-70.892,-58.650,60.679,150.3372,29.8340,0.0000
C00594=-74.369,-55.652,61.230,149.1322,12.7656,0.0000
C00595=-77.639,-55.369,62.625,172.6300,-2.5325,0.0000
C00596=-81.437,-56.971,64.575,-178.9120,0.5624,0.0000
C00597=-86.067,-59.672,66.618,-175.4330,2.6187,0.0000
C00598=-91.238,-62.811,68.213,-173.3819,3.6485,0.0000
C00599=-96.366,-65.383,69.012,-172.6286,1.9900,0.0000
C00600=-101.946,-65.289,69.436,-175.6250,-1.2614,0.0000
C00601=-107.195,-62.403,69.783,-178.2357,-1.5455,0.0000
C00602=-111.057,-57.205,70.135,-179.9328,-0.1261,0.0000
C00603=-114.095,-51.040,70.368,-179.9927,-0.0161,0.0000
C00604=-116.768,-44.586,70.368,-179.9938,-0.0165,0.0000
C00605=-118.979,-38.079,70.135,-179.9583,-0.1367,0.0000
C00606=-119.924,-31.673,69.783,179.8452,-2.3398,0.0000
C00607=-118.253,-25.920,69.436,177.7935,-3.9853,0.0000
C00608=-114.374,-21.908,69.012,173.3806,-3.8279,0.0000
C00609=-108.929,-20.101,68.213,172.7548,-2.1162,0.0000
C00610=-103.053,-18.664,66.618,174.9241,-1.3829,0.0000
C00611=-97.869,-17.300,64.575,178.8331,-0.3717,0.0000
C00612=-94.051,-15.748,62.625,-173.0028,3.4442,0.0000
C00613=-91.938,-13.235,61.230,-165.2938,30.2357,0.0000
C00614=-91.600,-8.656,60.679,179.8370,38.9469,0.0000
C00615=-91.854,-4.221,60.655,177.5938,39.2570,0.0000
C00616=-91.951,0.000,60.671,180.0000,39.2835,0.0000
C00617=-91.854,4.220,60.655,-177.5939,39.2571,0.0000
C00618=-91.600,8.656,60.679,-179.8394,38.9465,0.0000
C00619=-91.938,13.235,61.230,165.2943,30.2362,0.0000
C00620=-94.051,15.748,62.625,173.0028,3.4442,0.0000
C00621=-97.869,17.300,64.575,-178.8331,-0.3717,0.0000
C00622=-103.053,18.664,66.618,-174.9241,-1.3829,0.0000
C00623=-108.929,20.101,68.213,-172.7548,-2.1162,0.0000
C00624=-114.374,21.908,69.012,-173.3806,-3.8279,0.0000
C00625=-118.253,25.920,69.436,-177.7935,-3.9853,0.0000
C00626=-119.924,31.673,69.783,-179.8452,-2.3398,0.0000
C00627=-118.979,38.079,70.135,179.9583,-0.1367,0.0000
C00628=-116.768,44.586,70.368,179.9938,-0.0165,0.0000
C00629=-114.095,51.040,70.368,179.9927,-0.0161,0.0000
C00630=-111.057,57.205,70.135,179.9328,-0.1261,0.0000
C00631=-107.195,62.403,69.783,178.2357,-1.5455,0.0000
C00632=-101.946,65.289,69.436,175.6250,-1.2614,0.0000
C00633=-96.366,65.383,69.012,172.6286,1.9900,0.0000
C00634=-91.238,62.811,68.213,173.3819,3.6485,0.0000
C00635=-86.067,59.672,66.618,175.4330,2.6187,0.0000
C00636=-81.437,56.971,64.575,178.9120,0.5624,0.0000
C00637=-77.639,55.369,62.625,-172.6300,-2.5325,0.0000
C00638=-74.369,55.652,61.230,-149.1323,12.7648,0.0000
C00639=-70.891,58.650,60.679,-150.3382,29.8356,0.0000
C00640=-67.935,61.966,60.655,-151.2701,31.2824,0.0000
C00641=-65.019,65.019,60.671,-149.9541,30.0460,0.0000
C00642=-61.966,67.935,60.655,-148.7176,28.7300,0.0000
C00643=-58.650,70.892,60.679,-150.1660,29.6628,0.0000
C00644=-55.652,74.369,61.230,-167.2344,30.8678,0.0000
C00645=-55.369,77.639,62.625,177.4675,7.3700,0.0000
C00646=-56.971,81.437,64.575,-179.4376,-1.0880,0.0000
C00647=-59.672,86.067,66.618,-177.3813,-4.5670,0.0000
C00648=-62.811,91.238,68.213,-176.3515,-6.6181,0.0000
C00649=-65.383,96.366,69.012,-178.0100,-7.3714,0.0000
C00650=-65.289,101.946,69.436,178.7386,-4.3750,0.0000
C00651=-62.403,107.195,69.783,178.4545,-1.7643,0.0000
C00652=-57.205,111.057,70.135,179.8739,-0.0672,0.0000
C00653=-51.040,114.095,70.368,179.9839,-0.0073,0.0000
C00654=-44.586,116.768,70.368,179.9835,-0.0062,0.0000
C00655=-38.079,118.979,70.135,179.8633,-0.0417,0.0000
C00656=-31.673,119.924,69.783,177.6602,0.1548,0.0000
C00657=-25.920,118.253,69.436,176.0147,2.2065,0.0000
C00658=-21.908,114.374,69.012,176.1721,6.6194,0.0000
C00659=-20.101,108.929,68.213,177.8838,7.2452,0.0000
C00660=-18.664,103.053,66.618,178.6171,5.0759,0.0000
C00661=-17.300,97.869,64.575,179.6283,1.1669,0.0000
C00662=-15.748,94.051,62.625,-176.5558,-6.9972,0.0000
C00663=-13.235,91.938,61.230,-149.7638,-14.7057,0.0000
C00664=-8.656,91.600,60.679,-141.0535,0.1606,0.0000
C00665=-4.220,91.854,60.655,-140.7429,2.4061,0.0000
C00666=0.000,91.951,60.671,-140.7165,-0.0000,0.0000
C00667=0.000,90.559,62.374,-140.7584,-0.0001,0.0000
C00668=4.093,90.466,62.357,-140.7842,-2.3801,0.0000
C00669=8.442,90.224,62.382,-141.1213,0.1162,0.0000
C00670=12.972,90.607,62.961,-150.5794,15.1988,0.0000
C00671=15.425,92.833,64.428,-177.1997,6.1064,0.0000
C00672=16.927,96.833,66.479,179.4953,-1.6780,0.0000
C00673=18.257,102.257,68.628,178.6143,-5.3614,0.0000
C00674=19.662,108.407,70.305,177.9497,-7.4471,0.0000
C00675=21.431,114.114,71.144,176.2350,-6.8648,0.0000
C00676=25.471,118.199,71.589,175.9296,-2.3538,0.0000
C00677=31.317,119.989,71.953,177.6084,-0.1805,0.0000
C00678=37.853,119.054,72.323,179.8582,0.0430,0.0000
C00679=44.510,116.798,72.567,179.9830,0.0064,0.0000
C00680=51.115,114.062,72.567,179.9834,0.0075,0.0000
C00681=57.417,110.950,72.323,179.8693,0.0698,0.0000
C00682=62.701,106.989,71.953,178.4359,1.8192,0.0000
C00683=65.569,101.589,71.589,178.7825,4.5389,0.0000
C00684=65.537,95.845,71.144,-177.7897,7.5005,0.0000
C00685=62.752,90.559,70.305,-176.1604,6.7152,0.0000
C00686=59.397,85.216,68.628,-177.1801,4.7712,0.0000
C00687=56.501,80.440,66.479,-179.1701,1.5434,0.0000
C00688=54.736,76.550,64.428,177.6487,-6.2906,0.0000
C00689=54.896,73.242,62.961,-168.3232,-30.5776,0.0000
C00690=57.829,69.768,62.382,-150.3733,-29.7507,0.0000
C00691=61.075,66.864,62.357,-148.7667,-28.7067,0.0000
C00692=64.035,64.035,62.374,-149.9910,-30.0089,0.0000
C00693=66.864,61.075,62.357,-151.2933,-31.2334,0.0000
C00694=69.768,57.828,62.382,-150.2483,-29.6251,0.0000
C00695=73.242,54.896,62.961,-149.4223,-11.6775,0.0000
C00696=76.550,54.736,64.428,-173.7094,2.3513,0.0000
C00697=80.440,56.501,66.479,178.4566,-0.8299,0.0000
C00698=85.216,59.397,68.628,175.2288,-2.8199,0.0000
C00699=90.559,62.752,70.305,173.2848,-3.8396,0.0000
C00700=95.845,65.537,71.144,172.4995,-2.2103,0.0000
C00701=101.589,65.569,71.589,175.4611,1.2175,0.0000
C00702=106.989,62.701,71.953,178.1808,1.5641,0.0000
C00703=110.950,57.417,72.323,179.9302,0.1307,0.0000
C00704=114.062,51.115,72.567,179.9925,0.0166,0.0000
C00705=116.798,44.510,72.567,179.9936,0.0170,0.0000
C00706=119.054,37.853,72.323,179.9570,0.1418,0.0000
C00707=119.989,31.317,71.953,-179.8195,2.3916,0.0000
C00708=118.199,25.471,71.589,-177.6462,4.0704,0.0000
C00709=114.114,21.431,71.144,-173.1352,3.7650,0.0000
C00710=108.407,19.662,70.305,-172.5529,2.0503,0.0000
C00711=102.257,18.257,68.628,-174.6386,1.3857,0.0000
C00712=96.833,16.927,66.479,-178.3220,0.5047,0.0000
C00713=92.833,15.425,64.428,173.8936,-2.8003,0.0000
C00714=90.607,12.972,62.961,164.8012,-29.4206,0.0000
C00715=90.224,8.442,62.382,179.8838,-38.8787,0.0000
C00716=90.466,4.093,62.357,-177.6199,-39.2158,0.0000
C00717=90.559,0.000,62.374,-179.9999,-39.2416,0.0000
C00718=90.466,-4.093,62.357,177.6199,-39.2158,0.0000
C00719=90.224,-8.442,62.382,-179.8813,-38.8784,0.0000
C00720=90.607,-12.972,62.961,-164.8016,-29.4211,0.0000
C00721=92.833,-15.425,64.428,-173.8936,-2.8003,0.0000
C00722=96.833,-16.927,66.479,178.3220,0.5047,0.0000
C00723=102.257,-18.257,68.628,174.6386,1.3857,0.0000
C00724=108.407,-19.662,70.305,172.5529,2.0503,0.0000
C00725=114.114,-21.431,71.144,173.1352,3.7650,0.0000
C00726=118.199,-25.471,71.589,177.6462,4.0704,0.0000
C00727=119.989,-31.317,71.953,179.8195,2.3916,0.0000
C00728=119.054,-37.853,72.323,-179.9570,0.1418,0.0000
C00729=116.798,-44.510,72.567,-179.9936,0.0170,0.0000
C00730=114.062,-51.115,72.567,-179.9925,0.0166,0.0000
C00731=110.950,-57.417,72.323,-179.9302,0.1307,0.0000
C00732=106.989,-62.701,71.953,-178.1808,1.5641,0.0000
C00733=101.589,-65.569,71.589,-175.4611,1.2175,0.0000
C00734=95.845,-65.537,71.144,-172.4995,-2.2103,0.0000
C00735=90.559,-62.752,70.305,-173.2848,-3.8396,0.0000
C00736=85.216,-59.397,68.628,-175.2288,-2.8199,0.0000
C00737=80.440,-56.501,66.479,-178.4566,-0.8299,0.0000
C00738=76.550,-54.736,64.428,173.7094,2.3513,0.0000
C00739=73.242,-54.896,62.961,149.4224,-11.6768,0.0000
C00740=69.768,-57.829,62.382,150.2493,-29.6267,0.0000
C00741=66.864,-61.075,62.357,151.2933,-31.2333,0.0000
C00742=64.035,-64.035,62.374,149.9911,-30.0090,0.0000
C00743=61.075,-66.864,62.357,148.7666,-28.7067,0.0000
C00744=57.828,-69.768,62.382,150.3749,-29.7517,0.0000
C00745=54.896,-73.242,62.961,168.3225,-30.5777,0.0000
C00746=54.736,-76.550,64.428,-177.6487,-6.2906,0.0000
C00747=56.501,-80.440,66.479,179.1701,1.5434,0.0000
C00748=59.397,-85.216,68.628,177.1801,4.7712,0.0000
C00749=62.752,-90.559,70.305,176.1604,6.7152,0.0000
C00750=65.537,-95.845,71.144,177.7897,7.5005,0.0000
C00751=65.569,-101.589,71.589,-178.7825,4.5389,0.0000
C00752=62.701,-106.989,71.953,-178.4359,1.8192,0.0000
C00753=57.417,-110.950,72.323,-179.8693,0.0698,0.0000
C00754=51.115,-114.062,72.567,-179.9834,0.0075,0.0000
C00755=44.510,-116.798,72.567,-179.9830,0.0064,0.0000
C00756=37.853,-119.054,72.323,-179.8582,0.0430,0.0000
C00757=31.317,-119.989,71.953,-177.6084,-0.1805,0.0000
C00758=25.471,-118.199,71.589,-175.9296,-2.3538,0.0000
C00759=21.431,-114.114,71.144,-176.2350,-6.8648,0.0000
C00760=19.662,-108.407,70.305,-177.9497,-7.4471,0.0000
C00761=18.257,-102.257,68.628,-178.6143,-5.3614,0.0000
C00762=16.927,-96.833,66.479,-179.4953,-1.6780,0.0000
C00763=15.425,-92.833,64.428,177.1997,6.1064,0.0000
C00764=12.972,-90.607,62.961,150.5794,15.1988,0.0000
C00765=8.442,-90.224,62.382,141.1213,0.1162,0.0000
C00766=4.093,-90.466,62.357,140.7842,-2.3801,0.0000
C00767=0.000,-90.559,62.374,140.7584,-0.0001,0.0000
C00768=0.000,-90.559,62.374,140.7584,-0.0001,0.0000
C00769=-4.093,-90.466,62.357,140.7842,2.3801,0.0000
C00770=-8.442,-90.224,62.382,141.1216,-0.1187,0.0000
C00771=-12.972,-90.607,62.961,150.5789,-15.1984,0.0000
C00772=-15.425,-92.833,64.428,177.1997,-6.1064,0.0000
C00773=-16.927,-96.833,66.479,-179.4953,1.6780,0.0000
C00774=-18.257,-102.257,68.628,-178.6143,5.3614,0.0000
C00775=-19.662,-108.407,70.305,-177.9497,7.4471,0.0000
C00776=-21.431,-114.114,71.144,-176.2350,6.8648,0.0000
C00777=-25.471,-118.199,71.589,-175.9296,2.3538,0.0000
C00778=-31.317,-119.989,71.953,-177.6084,0.1805,0.0000
C00779=-37.853,-119.054,72.323,-179.8582,-0.0430,0.0000
C00780=-44.510,-116.798,72.567,-179.9830,-0.0064,0.0000
C00781=-51.115,-114.062,72.567,-179.9834,-0.0075,0.0000
C00782=-57.417,-110.950,72.323,-179.8693,-0.0698,0.0000
C00783=-62.701,-106.989,71.953,-178.4359,-1.8192,0.0000
C00784=-65.569,-101.589,71.589,-178.7825,-4.5389,0.0000
C00785=-65.537,-95.845,71.144,177.7897,-7.5005,0.0000
C00786=-62.752,-90.559,70.305,176.1604,-6.7152,0.0000
C00787=-59.397,-85.216,68.628,177.1801,-4.7712,0.0000
C00788=-56.501,-80.440,66.479,179.1701,-1.5434,0.0000
C00789=-54.736,-76.550,64.428,-177.6487,6.2906,0.0000
C00790=-54.896,-73.242,62.961,168.3232,30.5776,0.0000
C00791=-57.829,-69.768,62.382,150.3733,29.7507,0.0000
C00792=-61.075,-66.864,62.357,148.7667,28.7067,0.0000
C00793=-64.035,-64.035,62.374,149.9910,30.0089,0.0000
C00794=-66.864,-61.075,62.357,151.2933,31.2334,0.0000
C00795=-69.768,-57.828,62.382,150.2483,29.6251,0.0000
C00796=-73.242,-54.896,62.961,149.4223,11.6775,0.0000
C00797=-76.550,-54.736,64.428,173.7094,-2.3513,0.0000
C00798=-80.440,-56.501,66.479,-178.4566,0.8299,0.0000
C00799=-85.216,-59.397,68.628,-175.2288,2.8199,0.0000
C00800=-90.559,-62.752,70.305,-173.2848,3.8396,0.0000
C00801=-95.845,-65.537,71.144,-172.4995,2.2103,0.0000
C00802=-101.589,-65.569,71.589,-175.4611,-1.2175,0.0000
C00803=-106.989,-62.701,71.953,-178.1808,-1.5641,0.0000
C00804=-110.950,-57.417,72.323,-179.9302,-0.1307,0.0000
C00805=-114.062,-51.115,72.567,-179.9925,-0.0166,0.0000
C00806=-116.798,-44.510,72.567,-179.9936,-0.0170,0.0000
C00807=-119.054,-37.853,72.323,-179.9570,-0.1418,0.0000
C00808=-119.989,-31.317,71.953,179.8195,-2.3916,0.0000
C00809=-118.199,-25.471,71.589,177.6462,-4.0704,0.0000
C00810=-114.114,-21.431,71.144,173.1352,-3.7650,0.0000
C00811=-108.407,-19.662,70.305,172.5529,-2.0503,0.0000
C00812=-102.257,-18.257,68.628,174.6386,-1.3857,0.0000
C00813=-96.833,-16.927,66.479,178.3220,-0.5047,0.0000
C00814=-92.833,-15.425,64.428,-173.8936,2.8003,0.0000
C00815=-90.607,-12.972,62.961,-164.8012,29.4206,0.0000
C00816=-90.224,-8.442,62.382,-179.8838,38.8787,0.0000
C00817=-90.466,-4.093,62.357,177.6199,39.2158,0.0000
C00818=-90.559,0.000,62.374,179.9999,39.2416,0.0000
C00819=-90.466,4.093,62.357,-177.6199,39.2158,0.0000
C00820=-90.224,8.442,62.382,179.8813,38.8784,0.0000
C00821=-90.607,12.972,62.961,164.8016,29.4211,0.0000
C00822=-92.833,15.425,64.428,173.8936,2.8003,0.0000
C00823=-96.833,16.927,66.479,-178.3220,-0.5047,0.0000
C00824=-102.257,18.257,68.628,-174.6386,-1.3857,0.0000
C00825=-108.407,19.662,70.305,-172.5529,-2.0503,0.0000
C00826=-114.114,21.431,71.144,-173.1352,-3.7650,0.0000
C00827=-118.199,25.471,71.589,-177.6462,-4.0704,0.0000
C00828=-119.989,31.317,71.953,-179.8195,-2.3916,0.0000
C00829=-119.054,37.853,72.323,179.9570,-0.1418,0.0000
C00830=-116.798,44.510,72.567,179.9936,-0.0170,0.0000
C00831=-114.062,51.115,72.567,179.9925,-0.0166,0.0000
C00832=-110.950,57.417,72.323,179.9302,-0.1307,0.0000
C00833=-106.989,62.701,71.953,178.1808,-1.5641,0.0000
C00834=-101.589,65.569,71.589,175.4611,-1.2175,0.0000
C00835=-95.845,65.537,71.144,172.4995,2.2103,0.0000
C00836=-90.559,62.752,70.305,173.2848,3.8396,0.0000
C00837=-85.216,59.397,68.628,175.2288,2.8199,0.0000
C00838=-80.440,56.501,66.479,178.4566,0.8299,0.0000
C00839=-76.550,54.736,64.428,-173.7094,-2.3513,0.0000
C00840=-73.242,54.896,62.961,-149.4224,11.6768,0.0000
C00841=-69.768,57.829,62.382,-150.2493,29.6267,0.0000
C00842=-66.864,61.075,62.357,-151.2933,31.2333,0.0000
C00843=-64.035,64.035,62.374,-149.9911,30.0090,0.0000
C00844=-61.075,66.864,62.357,-148.7666,28.7067,0.0000
C00845=-57.828,69.768,62.382,-150.3749,29.7517,0.0000
C00846=-54.896,73.242,62.961,-168.3225,30.5777,0.0000
C00847=-54.736,76.550,64.428,177.6487,6.2906,0.0000
C00848=-56.501,80.440,66.479,-179.1701,-1.5434,0.0000
C00849=-59.397,85.216,68.628,-177.1801,-4.7712,0.0000
C00850=-62.752,90.559,70.305,-176.1604,-6.7152,0.0000
C00851=-65.537,95.845,71.144,-177.7897,-7.5005,0.0000
C00852=-65.569,101.589,71.589,178.7825,-4.5389,0.0000
C00853=-62.701,106.989,71.953,178.4359,-1.8192,0.0000
C00854=-57.417,110.950,72.323,179.8693,-0.0698,0.0000
C00855=-51.115,114.062,72.567,179.9834,-0.0075,0.0000
C00856=-44.510,116.798,72.567,179.9830,-0.0064,0.0000
C00857=-37.853,119.054,72.323,179.8582,-0.0430,0.0000
C00858=-31.317,119.989,71.953,177.6084,0.1805,0.0000
C00859=-25.471,118.199,71.589,175.9296,2.3538,0.0000
C00860=-21.431,114.114,71.144,176.2350,6.8648,0.0000
C00861=-19.662,108.407,70.305,177.9497,7.4471,0.0000
C00862=-18.257,102.257,68.628,178.6143,5.3614,0.0000
C00863=-16.927,96.833,66.479,179.4953,1.6780,0.0000
C00864=-15.425,92.833,64.428,-177.1997,-6.1064,0.0000
C00865=-12.972,90.607,62.961,-150.5789,-15.1984,0.0000
C00866=-8.442,90.224,62.382,-141.1216,-0.1187,0.0000
C00867=-4.093,90.466,62.357,-140.7842,2.3801,0.0000
C00868=0.000,90.559,62.374,-140.7584,-0.0001,0.0000
C00869=0.000,89.168,64.079,-140.8474,-0.0002,0.0000
C00870=3.966,89.081,64.061,-140.8726,-2.3488,0.0000
C00871=8.228,88.851,64.087,-141.2392,0.4004,0.0000
C00872=12.710,89.278,64.695,-151.4598,15.6079,0.0000
C00873=15.103,91.619,66.234,-177.7569,5.2402,0.0000
C00874=16.557,95.802,68.387,179.3909,-2.1400,0.0000
C00875=17.853,101.468,70.642,178.6238,-5.6002,0.0000
C00876=19.229,107.891,72.399,178.0238,-7.5977,0.0000
C00877=20.959,113.857,73.277,176.3191,-7.0565,0.0000
C00878=25.027,118.145,73.743,175.8732,-2.4841,0.0000
C00879=30.965,120.053,74.124,177.5702,-0.2049,0.0000
C00880=37.631,119.127,74.510,179.8541,0.0441,0.0000
C00881=44.434,116.827,74.765,179.9826,0.0065,0.0000
C00882=51.189,114.029,74.765,179.9831,0.0077,0.0000
C00883=57.626,110.845,74.510,179.8656,0.0720,0.0000
C00884=62.994,106.786,74.124,178.4261,1.8634,0.0000
C00885=65.845,101.238,73.743,178.8346,4.6704,0.0000
C00886=65.689,95.330,73.277,-177.5927,7.5770,0.0000
C00887=62.694,89.887,72.399,-176.0004,6.7704,0.0000
C00888=59.124,84.373,70.642,-177.0035,4.9336,0.0000
C00889=56.035,79.449,68.387,-178.9169,1.9439,0.0000
C00890=54.105,75.463,66.234,177.8721,-5.2875,0.0000
C00891=54.142,72.117,64.695,-169.4060,-30.2038,0.0000
C00892=57.009,68.645,64.087,-150.6296,-29.7986,0.0000
C00893=60.185,65.794,64.061,-148.8590,-28.6438,0.0000
C00894=63.052,63.052,64.079,-150.0696,-29.9302,0.0000
C00895=65.794,60.185,64.061,-151.3563,-31.1411,0.0000
C00896=68.645,57.008,64.087,-150.2004,-29.3687,0.0000
C00897=72.117,54.142,64.695,-149.7960,-10.5946,0.0000
C00898=75.463,54.105,66.234,-174.7125,2.1279,0.0000
C00899=79.449,56.035,68.387,178.0561,-1.0831,0.0000
C00900=84.373,59.124,70.642,175.0664,-2.9965,0.0000
C00901=89.887,62.694,72.399,173.2296,-3.9996,0.0000
C00902=95.330,65.689,73.277,172.4230,-2.4073,0.0000
C00903=101.238,65.845,73.743,175.3296,1.1654,0.0000
C00904=106.786,62.994,74.124,178.1366,1.5739,0.0000
C00905=110.845,57.626,74.510,179.9280,0.1344,0.0000
C00906=114.029,51.189,74.765,179.9923,0.0169,0.0000
C00907=116.827,44.434,74.765,179.9935,0.0174,0.0000
C00908=119.127,37.631,74.510,179.9559,0.1459,0.0000
C00909=120.053,30.965,74.124,-179.7951,2.4298,0.0000
C00910=118.145,25.027,73.743,-177.5159,4.1268,0.0000
C00911=113.857,20.959,73.277,-172.9435,3.6809,0.0000
C00912=107.891,19.229,72.399,-172.4023,1.9762,0.0000
C00913=101.468,17.853,70.642,-174.3998,1.3762,0.0000
C00914=95.802,16.557,68.387,-177.8600,0.6091,0.0000
C00915=91.619,15.103,66.234,174.7598,-2.2431,0.0000
C00916=89.278,12.710,64.695,164.3921,-28.5402,0.0000
C00917=88.851,8.228,64.087,179.5996,-38.7608,0.0000
C00918=89.081,3.966,64.061,-177.6512,-39.1274,0.0000
C00919=89.168,0.000,64.079,-179.9998,-39.1526,0.0000
C00920=89.081,-3.966,64.061,177.6511,-39.1275,0.0000
C00921=88.851,-8.229,64.087,-179.5971,-38.7604,0.0000
C00922=89.278,-12.710,64.695,-164.3924,-28.5406,0.0000
C00923=91.619,-15.103,66.234,-174.7598,-2.2431,0.0000
C00924=95.802,-16.557,68.387,177.8600,0.6091,0.0000
C00925=101.468,-17.853,70.642,174.3998,1.3762,0.0000
C00926=107.891,-19.229,72.399,172.4023,1.9762,0.0000
C00927=113.857,-20.959,73.277,172.9435,3.6809,0.0000
C00928=118.145,-25.027,73.743,177.5159,4.1268,0.0000
C00929=120.053,-30.965,74.124,179.7951,2.4298,0.0000
C00930=119.127,-37.631,74.510,-179.9559,0.1459,0.0000
C00931=116.827,-44.434,74.765,-179.9935,0.0174,0.0000
C00932=114.029,-51.189,74.765,-179.9923,0.0169,0.0000
C00933=110.845,-57.626,74.510,-179.9280,0.1344,0.0000
C00934=106.786,-62.994,74.124,-178.1366,1.5739,0.0000
C00935=101.238,-65.845,73.743,-175.3296,1.1654,0.0000
C00936=95.330,-65.689,73.277,-172.4230,-2.4073,0.0000
C00937=89.887,-62.694,72.399,-173.2296,-3.9996,0.0000
C00938=84.373,-59.124,70.642,-175.0664,-2.9965,0.0000
C00939=79.449,-56.035,68.387,-178.0561,-1.0831,0.0000
C00940=75.463,-54.105,66.234,174.7125,2.1279,0.0000
C00941=72.117,-54.142,64.695,149.7962,-10.5940,0.0000
C00942=68.645,-57.009,64.087,150.2014,-29.3704,0.0000
C00943=65.794,-60.185,64.061,151.3562,-31.1410,0.0000
C00944=63.052,-63.052,64.079,150.0698,-29.9304,0.0000
C00945=60.185,-65.794,64.061,148.8589,-28.6437,0.0000
C00946=57.008,-68.645,64.087,150.6313,-29.7996,0.0000
C00947=54.142,-72.117,64.695,169.4054,-30.2040,0.0000
C00948=54.105,-75.463,66.234,-177.8721,-5.2875,0.0000
C00949=56.035,-79.449,68.387,178.9169,1.9439,0.0000
C00950=59.124,-84.373,70.642,177.0035,4.9336,0.0000
C00951=62.694,-89.887,72.399,176.0004,6.7704,0.0000
C00952=65.689,-95.330,73.277,177.5927,7.5770,0.0000
C00953=65.845,-101.238,73.743,-178.8346,4.6704,0.0000
C00954=62.994,-106.786,74.124,-178.4261,1.8634,0.0000
C00955=57.626,-110.845,74.510,-179.8656,0.0720,0.0000
C00956=51.189,-114.029,74.765,-179.9831,0.0077,0.0000
C00957=44.434,-116.827,74.765,-179.9826,0.0065,0.0000
C00958=37.631,-119.127,74.510,-179.8541,0.0441,0.0000
C00959=30.965,-120.053,74.124,-177.5702,-0.2049,0.0000
C00960=25.027,-118.145,73.743,-175.8732,-2.4841,0.0000
C00961=20.959,-113.857,73.277,-176.3191,-7.0565,0.0000
C00962=19.229,-107.891,72.399,-178.0238,-7.5977,0.0000
C00963=17.853,-101.468,70.642,-178.6238,-5.6002,0.0000
C00964=16.557,-95.802,68.387,-179.3909,-2.1400,0.0000
C00965=15.103,-91.619,66.234,177.7569,5.2402,0.0000
C00966=12.710,-89.278,64.695,151.4598,15.6079,0.0000
C00967=8.228,-88.851,64.087,141.2392,0.4004,0.0000
C00968=3.966,-89.081,64.061,140.8726,-2.3488,0.0000
C00969=0.000,-89.168,64.079,140.8474,-0.0002,0.0000
C00970=0.000,-89.168,64.079,140.8474,-0.0002,0.0000
C00971=-3.966,-89.081,64.061,140.8725,2.3489,0.0000
C00972=-8.229,-88.851,64.087,141.2396,-0.4029,0.0000
C00973=-12.710,-89.278,64.695,151.4594,-15.6076,0.0000
C00974=-15.103,-91.619,66.234,177.7569,-5.2402,0.0000
C00975=-16.557,-95.802,68.387,-179.3909,2.1400,0.0000
C00976=-17.853,-101.468,70.642,-178.6238,5.6002,0.0000
C00977=-19.229,-107.891,72.399,-178.0238,7.5977,0.0000
C00978=-20.959,-113.857,73.277,-176.3191,7.0565,0.0000
C00979=-25.027,-118.145,73.743,-175.8732,2.4841,0.0000
C00980=-30.965,-120.053,74.124,-177.5702,0.2049,0.0000
C00981=-37.631,-119.127,74.510,-179.8541,-0.0441,0.0000
C00982=-44.434,-116.827,74.765,-179.9826,-0.0065,0.0000
C00983=-51.189,-114.029,74.765,-179.9831,-0.0077,0.0000
C00984=-57.626,-110.845,74.510,-179.8656,-0.0720,0.0000
C00985=-62.994,-106.786,74.124,-178.4261,-1.8634,0.0000
C00986=-65.845,-101.238,73.743,-178.8346,-4.6704,0.0000
C00987=-65.689,-95.330,73.277,177.5927,-7.5770,0.0000
C00988=-62.694,-89.887,72.399,176.0004,-6.7704,0.0000
C00989=-59.124,-84.373,70.642,177.0035,-4.9336,0.0000
C00990=-56.035,-79.449,68.387,178.9169,-1.9439,0.0000
C00991=-54.105,-75.463,66.234,-177.8721,5.2875,0.0000
C00992=-54.142,-72.117,64.695,169.4060,30.2038,0.0000
C00993=-57.009,-68.645,64.087,150.6296,29.7986,0.0000
C00994=-60.185,-65.794,64.061,148.8590,28.6438,0.0000
C00995=-63.052,-63.052,64.079,150.0696,29.9302,0.0000
C00996=-65.794,-60.185,64.061,151.3563,31.1411,0.0000
C00997=-68.645,-57.008,64.087,150.2004,29.3687,0.0000
C00998=-72.117,-54.142,64.695,149.7960,10.5946,0.0000
C00999=-75.463,-54.105,66.234,174.7125,-2.1279,0.0000
C01000=-79.449,-56.035,68.387,-178.0561,1.0831,0.0000
C01001=-84.373,-59.124,70.642,-175.0664,2.9965,0.0000
C01002=-89.887,-62.694,72.399,-173.2296,3.9996,0.0000
C01003=-95.330,-65.689,73.277,-172.4230,2.4073,0.0000
C01004=-101.238,-65.845,73.743,-175.3296,-1.1654,0.0000
C01005=-106.786,-62.994,74.124,-178.1366,-1.5739,0.0000
C01006=-110.845,-57.626,74.510,-179.9280,-0.1344,0.0000
C01007=-114.029,-51.189,74.765,-179.9923,-0.0169,0.0000
C01008=-116.827,-44.434,74.765,-179.9935,-0.0174,0.0000
C01009=-119.127,-37.631,74.510,-179.9559,-0.1459,0.0000
C01010=-120.053,-30.965,74.124,179.7951,-2.4298,0.0000
C01011=-118.145,-25.027,73.743,177.5159,-4.1268,0.0000
C01012=-113.857,-20.959,73.277,172.9435,-3.6809,0.0000
C01013=-107.891,-19.229,72.399,172.4023,-1.9762,0.0000
C01014=-101.468,-17.853,70.642,174.3998,-1.3762,0.0000
C01015=-95.802,-16.557,68.387,177.8600,-0.6091,0.0000
C01016=-91.619,-15.103,66.234,-174.7598,2.2431,0.0000
C01017=-89.278,-12.710,64.695,-164.3921,28.5402,0.0000
C01018=-88.851,-8.228,64.087,-179.5996,38.7608,0.0000
C01019=-89.081,-3.966,64.061,177.6512,39.1274,0.0000
C01020=-89.168,0.000,64.079,179.9998,39.1526,0.0000
C01021=-89.081,3.966,64.061,-177.6511,39.1275,0.0000
C01022=-88.851,8.229,64.087,179.5971,38.7604,0.0000
C01023=-89.278,12.710,64.695,164.3924,28.5406,0.0000
C01024=-91.619,15.103,66.234,174.7598,2.2431,0.0000
C01025=-95.802,16.557,68.387,-177.8600,-0.6091,0.0000
C01026=-101.468,17.853,70.642,-174.3998,-1.3762,0.0000
C01027=-107.891,19.229,72.399,-172.4023,-1.9762,0.0000
C01028=-113.857,20.959,73.277,-172.9435,-3.6809,0.0000
C01029=-118.145,25.027,73.743,-177.5159,-4.1268,0.0000
C01030=-120.053,30.965,74.124,-179.7951,-2.4298,0.0000
C01031=-119.127,37.631,74.510,179.9559,-0.1459,0.0000
C01032=-116.827,44.434,74.765,179.9935,-0.0174,0.0000
C01033=-114.029,51.189,74.765,179.9923,-0.0169,0.0000
C01034=-110.845,57.626,74.510,179.9280,-0.1344,0.0000
C01035=-106.786,62.994,74.124,178.1366,-1.5739,0.0000
C01036=-101.238,65.845,73.743,175.3296,-1.1654,0.0000
C01037=-95.330,65.689,73.277,172.4230,2.4073,0.0000
C01038=-89.887,62.694,72.399,173.2296,3.9996,0.0000
C01039=-84.373,59.124,70.642,175.0664,2.9965,0.0000
C01040=-79.449,56.035,68.387,178.0561,1.0831,0.0000
C01041=-75.463,54.105,66.234,-174.7125,-2.1279,0.0000
C01042=-72.117,54.142,64.695,-149.7962,10.5940,0.0000
C01043=-68.645,57.009,64.087,-150.2014,29.3704,0.0000
C01044=-65.794,60.185,64.061,-151.3562,31.1410,0.0000
C01045=-63.052,63.052,64.079,-150.0698,29.9304,0.0000
C01046=-60.185,65.794,64.061,-148.8589,28.6437,0.0000
C01047=-57.008,68.645,64.087,-150.6313,29.7996,0.0000
C01048=-54.142,72.117,64.695,-169.4054,30.2040,0.0000
C01049=-54.105,75.463,66.234,177.8721,5.2875,0.0000
C01050=-56.035,79.449,68.387,-178.9169,-1.9439,0.0000
C01051=-59.124,84.373,70.642,-177.0035,-4.9336,0.0000
C01052=-62.694,89.887,72.399,-176.0004,-6.7704,0.0000
C01053=-65.689,95.330,73.277,-177.5927,-7.5770,0.0000
C01054=-65.845,101.238,73.743,178.8346,-4.6704,0.0000
C01055=-62.994,106.786,74.124,178.4261,-1.8634,0.0000
C01056=-57.626,110.845,74.510,179.8656,-0.0720,0.0000
C01057=-51.189,114.029,74.765,179.9831,-0.0077,0.0000
C01058=-44.434,116.827,74.765,179.9826,-0.0065,0.0000
C01059=-37.631,119.127,74.510,179.8541,-0.0441,0.0000
C01060=-30.965,120.053,74.124,177.5702,0.2049,0.0000
C01061=-25.027,118.145,73.743,175.8732,2.4841,0.0000
C01062=-20.959,113.857,73.277,176.3191,7.0565,0.0000
C01063=-19.229,107.891,72.399,178.0238,7.5977,0.0000
C01064=-17.853,101.468,70.642,178.6238,5.6002,0.0000
C01065=-16.557,95.802,68.387,179.3909,2.1400,0.0000
C01066=-15.103,91.619,66.234,-177.7569,-5.2402,0.0000
C01067=-12.710,89.278,64.695,-151.4594,-15.6076,0.0000
C01068=-8.229,88.851,64.087,-141.2396,-0.4029,0.0000
C01069=-3.966,89.081,64.061,-140.8725,2.3489,0.0000
C01070=0.000,89.168,64.079,-140.8474,-0.0002,0.0000
C01071=0.000,87.781,65.786,-140.9841,-0.0003,0.0000
C01072=3.840,87.698,65.768,-141.0086,-2.3123,0.0000
C01073=8.015,87.481,65.795,-141.4076,0.6879,0.0000
C01074=12.449,87.954,66.432,-152.3994,15.9319,0.0000
C01075=14.782,90.410,68.045,-178.2360,4.4069,0.0000
C01076=16.189,94.778,70.299,179.3108,-2.5536,0.0000
C01077=17.454,100.687,72.659,178.6435,-5.7935,0.0000
C01078=18.801,107.381,74.496,178.1038,-7.6987,0.0000
C01079=20.495,113.605,75.413,176.4208,-7.1953,0.0000
C01080=24.591,118.093,75.899,175.8447,-2.5954,0.0000
C01081=30.620,120.116,76.296,177.5461,-0.2275,0.0000
C01082=37.413,119.199,76.698,179.8510,0.0449,0.0000
C01083=44.361,116.855,76.964,179.9823,0.0066,0.0000
C01084=51.261,113.997,76.964,179.9828,0.0078,0.0000
C01085=57.831,110.742,76.698,179.8629,0.0736,0.0000
C01086=63.283,106.586,76.296,178.4250,1.8965,0.0000
C01087=66.116,100.892,75.899,178.8932,4.7688,0.0000
C01088=65.838,94.823,75.413,-177.4212,7.6040,0.0000
C01089=62.636,89.224,74.496,-175.8716,6.7862,0.0000
C01090=58.855,83.538,72.659,-176.8519,5.0569,0.0000
C01091=55.571,78.465,70.299,-178.6807,2.2930,0.0000
C01092=53.477,74.382,68.045,178.1261,-4.3616,0.0000
C01093=53.390,70.995,66.432,-170.4731,-29.7491,0.0000
C01094=56.191,67.526,65.795,-150.9333,-29.8046,0.0000
C01095=59.297,64.727,65.768,-148.9949,-28.5407,0.0000
C01096=62.071,62.071,65.786,-150.1902,-29.8095,0.0000
C01097=64.727,59.297,65.768,-151.4594,-31.0052,0.0000
C01098=67.526,56.190,65.795,-150.1944,-29.0650,0.0000
C01099=70.995,53.390,66.432,-150.2508,-9.5275,0.0000
C01100=74.382,53.477,68.045,-175.6384,1.8739,0.0000
C01101=78.465,55.571,70.299,177.7070,-1.3193,0.0000
C01102=83.538,58.855,72.659,174.9431,-3.1481,0.0000
C01103=89.224,62.636,74.496,173.2138,-4.1284,0.0000
C01104=94.823,65.838,75.413,172.3960,-2.5788,0.0000
C01105=100.892,66.116,75.899,175.2312,1.1068,0.0000
C01106=106.586,63.283,76.296,178.1035,1.5750,0.0000
C01107=110.742,57.831,76.698,179.9264,0.1371,0.0000
C01108=113.997,51.261,76.964,179.9922,0.0172,0.0000
C01109=116.855,44.361,76.964,179.9934,0.0177,0.0000
C01110=119.199,37.413,76.698,179.9551,0.1490,0.0000
C01111=120.116,30.620,76.296,-179.7725,2.4539,0.0000
C01112=118.093,24.591,75.899,-177.4046,4.1553,0.0000
C01113=113.605,20.495,75.413,-172.8047,3.5792,0.0000
C01114=107.381,18.801,74.496,-172.3013,1.8962,0.0000
C01115=100.687,17.454,72.659,-174.2065,1.3565,0.0000
C01116=94.778,16.189,70.299,-177.4464,0.6892,0.0000
C01117=90.410,14.782,68.045,175.5931,-1.7640,0.0000
C01118=87.954,12.449,66.432,164.0681,-27.6006,0.0000
C01119=87.481,8.015,65.795,179.3121,-38.5924,0.0000
C01120=87.698,3.840,65.768,-177.6877,-38.9914,0.0000
C01121=87.781,0.000,65.786,-179.9997,-39.0159,0.0000
C01122=87.698,-3.839,65.768,177.6874,-38.9915,0.0000
C01123=87.481,-8.015,65.795,-179.3096,-38.5920,0.0000
C01124=87.954,-12.449,66.432,-164.0683,-27.6010,0.0000
C01125=90.410,-14.782,68.045,-175.5931,-1.7640,0.0000
C01126=94.778,-16.189,70.299,177.4464,0.6892,0.0000
C01127=100.687,-17.454,72.659,174.2065,1.3565,0.0000
C01128=107.381,-18.801,74.496,172.3013,1.8962,0.0000
C01129=113.605,-20.495,75.413,172.8047,3.5792,0.0000
C01130=118.093,-24.591,75.899,177.4046,4.1553,0.0000
C01131=120.116,-30.620,76.296,179.7725,2.4539,0.0000
C01132=119.199,-37.413,76.698,-179.9551,0.1490,0.0000
C01133=116.855,-44.361,76.964,-179.9934,0.0177,0.0000
C01134=113.997,-51.261,76.964,-179.9922,0.0172,0.0000
C01135=110.742,-57.831,76.698,-179.9264,0.1371,0.0000
C01136=106.586,-63.283,76.296,-178.1035,1.5750,0.0000
C01137=100.892,-66.116,75.899,-175.2312,1.1068,0.0000
C01138=94.823,-65.838,75.413,-172.3960,-2.5788,0.0000
C01139=89.224,-62.636,74.496,-173.2138,-4.1284,0.0000
C01140=83.538,-58.855,72.659,-174.9431,-3.1481,0.0000
C01141=78.465,-55.571,70.299,-177.7070,-1.3193,0.0000
C01142=74.382,-53.477,68.045,175.6384,1.8739,0.0000
C01143=70.995,-53.390,66.432,150.2509,-9.5269,0.0000
C01144=67.526,-56.191,65.795,150.1954,-29.0667,0.0000
C01145=64.727,-59.297,65.768,151.4593,-31.0051,0.0000
C01146=62.071,-62.071,65.786,150.1905,-29.8098,0.0000
C01147=59.297,-64.727,65.768,148.9948,-28.5406,0.0000
C01148=56.190,-67.526,65.795,150.9350,-29.8056,0.0000
C01149=53.390,-70.995,66.432,170.4725,-29.7492,0.0000
C01150=53.477,-74.382,68.045,-178.1261,-4.3616,0.0000
C01151=55.571,-78.465,70.299,178.6807,2.2930,0.0000
C01152=58.855,-83.538,72.659,176.8519,5.0569,0.0000
C01153=62.636,-89.224,74.496,175.8716,6.7862,0.0000
C01154=65.838,-94.823,75.413,177.4212,7.6040,0.0000
C01155=66.116,-100.892,75.899,-178.8932,4.7688,0.0000
C01156=63.283,-106.586,76.296,-178.4250,1.8965,0.0000
C01157=57.831,-110.742,76.698,-179.8629,0.0736,0.0000
C01158=51.261,-113.997,76.964,-179.9828,0.0078,0.0000
C01159=44.361,-116.855,76.964,-179.9823,0.0066,0.0000
C01160=37.413,-119.199,76.698,-179.8510,0.0449,0.0000
C01161=30.620,-120.116,76.296,-177.5461,-0.2275,0.0000
C01162=24.591,-118.093,75.899,-175.8447,-2.5954,0.0000
C01163=20.495,-113.605,75.413,-176.4208,-7.1953,0.0000
C01164=18.801,-107.381,74.496,-178.1038,-7.6987,0.0000
C01165=17.454,-100.687,72.659,-178.6435,-5.7935,0.0000
C01166=16.189,-94.778,70.299,-179.3108,-2.5536,0.0000
C01167=14.782,-90.410,68.045,178.2360,4.4069,0.0000
C01168=12.449,-87.954,66.432,152.3994,15.9319,0.0000
C01169=8.015,-87.481,65.795,141.4076,0.6879,0.0000
C01170=3.840,-87.698,65.768,141.0086,-2.3123,0.0000
C01171=0.000,-87.781,65.786,140.9841,-0.0003,0.0000
C01172=0.000,-87.781,65.786,140.9841,-0.0003,0.0000
C01173=-3.839,-87.698,65.768,141.0085,2.3126,0.0000
C01174=-8.015,-87.481,65.795,141.4080,-0.6904,0.0000
C01175=-12.449,-87.954,66.432,152.3990,-15.9317,0.0000
C01176=-14.782,-90.410,68.045,178.2360,-4.4069,0.0000
C01177=-16.189,-94.778,70.299,-179.3108,2.5536,0.0000
C01178=-17.454,-100.687,72.659,-178.6435,5.7935,0.0000
C01179=-18.801,-107.381,74.496,-178.1038,7.6987,0.0000
C01180=-20.495,-113.605,75.413,-176.4208,7.1953,0.0000
C01181=-24.591,-118.093,75.899,-175.8447,2.5954,0.0000
C01182=-30.620,-120.116,76.296,-177.5461,0.2275,0.0000
C01183=-37.413,-119.199,76.698,-179.8510,-0.0449,0.0000
C01184=-44.361,-116.855,76.964,-179.9823,-0.0066,0.0000
C01185=-51.261,-113.997,76.964,-179.9828,-0.0078,0.0000
C01186=-57.831,-110.742,76.698,-179.8629,-0.0736,0.0000
C01187=-63.283,-106.586,76.296,-178.4250,-1.8965,0.0000
C01188=-66.116,-100.892,75.899,-178.8932,-4.7688,0.0000
C01189=-65.838,-94.823,75.413,177.4212,-7.6040,0.0000
C01190=-62.636,-89.224,74.496,175.8716,-6.7862,0.0000
C01191=-58.855,-83.538,72.659,176.8519,-5.0569,0.0000
C01192=-55.571,-78.465,70.299,178.6807,-2.2930,0.0000
C01193=-53.477,-74.382,68.045,-178.1261,4.3616,0.0000
C01194=-53.390,-70.995,66.432,170.4731,29.7491,0.0000
C01195=-56.191,-67.526,65.795,150.9333,29.8046,0.0000
C01196=-59.297,-64.727,65.768,148.9949,28.5407,0.0000
C01197=-62.071,-62.071,65.786,150.1902,29.8095,0.0000
C01198=-64.727,-59.297,65.768,151.4594,31.0052,0.0000
C01199=-67.526,-56.190,65.795,150.1944,29.0650,0.0000
C01200=-70.995,-53.390,66.432,150.2508,9.5275,0.0000
C01201=-74.382,-53.477,68.045,175.6384,-1.8739,0.0000
C01202=-78.465,-55.571,70.299,-177.7070,1.3193,0.0000
C01203=-83.538,-58.855,72.659,-174.9431,3.1481,0.0000
C01204=-89.224,-62.636,74.496,-173.2138,4.1284,0.0000
C01205=-94.823,-65.838,75.413,-172.3960,2.5788,0.0000
C01206=-100.892,-66.116,75.899,-175.2312,-1.1068,0.0000
C01207=-106.586,-63.283,76.296,-178.1035,-1.5750,0.0000
C01208=-110.742,-57.831,76.698,-179.9264,-0.1371,0.0000
C01209=-113.997,-51.261,76.964,-179.9922,-0.0172,0.0000
C01210=-116.855,-44.361,76.964,-179.9934,-0.0177,0.0000
C01211=-119.199,-37.413,76.698,-179.9551,-0.1490,0.0000
C01212=-120.116,-30.620,76.296,179.7725,-2.4539,0.0000
C01213=-118.093,-24.591,75.899,177.4046,-4.1553,0.0000
C01214=-113.605,-20.495,75.413,172.8047,-3.5792,0.0000
C01215=-107.381,-18.801,74.496,172.3013,-1.8962,0.0000
C01216=-100.687,-17.454,72.659,174.2065,-1.3565,0.0000
C01217=-94.778,-16.189,70.299,177.4464,-0.6892,0.0000
C01218=-90.410,-14.782,68.045,-175.5931,1.7640,0.0000
C01219=-87.954,-12.449,66.432,-164.0681,27.6006,0.0000
C01220=-87.481,-8.015,65.795,-179.3121,38.5924,0.0000
C01221=-87.698,-3.840,65.768,177.6877,38.9914,0.0000
C01222=-87.781,0.000,65.786,179.9997,39.0159,0.0000
C01223=-87.698,3.839,65.768,-177.6874,38.9915,0.0000
C01224=-87.481,8.015,65.795,179.3096,38.5920,0.0000
C01225=-87.954,12.449,66.432,164.0683,27.6010,0.0000
C01226=-90.410,14.782,68.045,175.5931,1.7640,0.0000
C01227=-94.778,16.189,70.299,-177.4464,-0.6892,0.0000
C01228=-100.687,17.454,72.659,-174.2065,-1.3565,0.0000
C01229=-107.381,18.801,74.496,-172.3013,-1.8962,0.0000
C01230=-113.605,20.495,75.413,-172.8047,-3.5792,0.0000
C01231=-118.093,24.591,75.899,-177.4046,-4.1553,0.0000
C01232=-120.116,30.620,76.296,-179.7725,-2.4539,0.0000
C01233=-119.199,37.413,76.698,179.9551,-0.1490,0.0000
C01234=-116.855,44.361,76.964,179.9934,-0.0177,0.0000
C01235=-113.997,51.261,76.964,179.9922,-0.0172,0.0000
C01236=-110.742,57.831,76.698,179.9264,-0.1371,0.0000
C01237=-106.586,63.283,76.296,178.1035,-1.5750,0.0000
C01238=-100.892,66.116,75.899,175.2312,-1.1068,0.0000
C01239=-94.823,65.838,75.413,172.3960,2.5788,0.0000
C01240=-89.224,62.636,74.496,173.2138,4.1284,0.0000
C01241=-83.538,58.855,72.659,174.9431,3.1481,0.0000
C01242=-78.465,55.571,70.299,177.7070,1.3193,0.0000
C01243=-74.382,53.477,68.045,-175.6384,-1.8739,0.0000
C01244=-70.995,53.390,66.432,-150.2509,9.5269,0.0000
C01245=-67.526,56.191,65.795,-150.1954,29.0667,0.0000
C01246=-64.727,59.297,65.768,-151.4593,31.0051,0.0000
C01247=-62.071,62.071,65.786,-150.1905,29.8098,0.0000
C01248=-59.297,64.727,65.768,-148.9948,28.5406,0.0000
C01249=-56.190,67.526,65.795,-150.9350,29.8056,0.0000
C01250=-53.390,70.995,66.432,-170.4725,29.7492,0.0000
C01251=-53.477,74.382,68.045,178.1261,4.3616,0.0000
C01252=-55.571,78.465,70.299,-178.6807,-2.2930,0.0000
C01253=-58.855,83.538,72.659,-176.8519,-5.0569,0.0000
C01254=-62.636,89.224,74.496,-175.8716,-6.7862,0.0000
C01255=-65.838,94.823,75.413,-177.4212,-7.6040,0.0000
C01256=-66.116,100.892,75.899,178.8932,-4.7688,0.0000
C01257=-63.283,106.586,76.296,178.4250,-1.8965,0.0000
C01258=-57.831,110.742,76.698,179.8629,-0.0736,0.0000
C01259=-51.261,113.997,76.964,179.9828,-0.0078,0.0000
C01260=-44.361,116.855,76.964,179.9823,-0.0066,0.0000
C01261=-37.413,119.199,76.698,179.8510,-0.0449,0.0000
C01262=-30.620,120.116,76.296,177.5461,0.2275,0.0000
C01263=-24.591,118.093,75.899,175.8447,2.5954,0.0000
C01264=-20.495,113.605,75.413,176.4208,7.1953,0.0000
C01265=-18.801,107.381,74.496,178.1038,7.6987,0.0000
C01266=-17.454,100.687,72.659,178.6435,5.7935,0.0000
C01267=-16.189,94.778,70.299,179.3108,2.5536,0.0000
C01268=-14.782,90.410,68.045,-178.2360,-4.4069,0.0000
C01269=-12.449,87.954,66.432,-152.3990,-15.9317,0.0000
C01270=-8.015,87.481,65.795,-141.4080,-0.6904,0.0000
C01271=-3.839,87.698,65.768,-141.0085,2.3126,0.0000
C01272=0.000,87.781,65.786,-140.9841,-0.0003,0.0000
C01273=0.000,86.399,67.498,-141.1694,-0.0003,0.0000
C01274=3.713,86.321,67.479,-141.1931,-2.2708,0.0000
C01275=7.803,86.115,67.507,-141.6274,0.9768,0.0000
C01276=12.189,86.634,68.173,-153.3915,16.1700,0.0000
C01277=14.463,89.208,69.859,-178.6452,3.6131,0.0000
C01278=15.824,93.763,72.217,179.2513,-2.9196,0.0000
C01279=17.059,99.916,74.682,178.6715,-5.9428,0.0000
C01280=18.380,106.881,76.596,178.1883,-7.7516,0.0000
C01281=20.040,113.357,77.551,176.5369,-7.2819,0.0000
C01282=24.163,118.041,78.056,175.8432,-2.6864,0.0000
C01283=30.282,120.177,78.469,177.5362,-0.2480,0.0000
C01284=37.200,119.269,78.887,179.8490,0.0453,0.0000
C01285=44.288,116.883,79.163,179.9821,0.0067,0.0000
C01286=51.332,113.965,79.163,179.9826,0.0079,0.0000
C01287=58.031,110.641,78.887,179.8612,0.0747,0.0000
C01288=63.566,106.390,78.469,178.4325,1.9179,0.0000
C01289=66.382,100.553,78.056,178.9566,4.8339,0.0000
C01290=65.985,94.325,77.551,-177.2768,7.5841,0.0000
C01291=62.579,88.573,76.596,-175.7743,6.7648,0.0000
C01292=58.589,82.714,74.682,-176.7258,5.1430,0.0000
C01293=55.112,77.490,72.217,-178.4635,2.5939,0.0000
C01294=52.853,73.307,69.859,178.4003,-3.5119,0.0000
C01295=52.641,69.878,68.173,-171.5145,-29.2163,0.0000
C01296=55.375,66.410,67.507,-151.2844,-29.7675,0.0000
C01297=58.412,63.664,67.479,-149.1751,-28.3970,0.0000
C01298=61.093,61.093,67.498,-150.3534,-29.6462,0.0000
C01299=63.663,58.413,67.479,-151.6031,-30.8251,0.0000
C01300=66.410,55.375,67.507,-150.2315,-28.7138,0.0000
C01301=69.878,52.641,68.173,-150.7835,-8.4859,0.0000
C01302=73.307,52.853,69.859,-176.4881,1.5997,0.0000
C01303=77.490,55.112,72.217,177.4061,-1.5365,0.0000
C01304=82.714,58.589,74.682,174.8570,-3.2742,0.0000
C01305=88.573,62.579,76.596,173.2352,-4.2257,0.0000
C01306=94.325,65.985,77.551,172.4159,-2.7232,0.0000
C01307=100.553,66.382,78.056,175.1661,1.0434,0.0000
C01308=106.390,63.566,78.469,178.0821,1.5675,0.0000
C01309=110.641,58.031,78.887,179.9253,0.1388,0.0000
C01310=113.965,51.332,79.163,179.9921,0.0174,0.0000
C01311=116.883,44.288,79.163,179.9933,0.0179,0.0000
C01312=119.269,37.200,78.887,179.9547,0.1510,0.0000
C01313=120.177,30.282,78.469,-179.7520,2.4638,0.0000
C01314=118.041,24.163,78.056,-177.3136,4.1568,0.0000
C01315=113.357,20.040,77.551,-172.7181,3.4631,0.0000
C01316=106.881,18.380,76.596,-172.2484,1.8117,0.0000
C01317=99.916,17.059,74.682,-174.0572,1.3285,0.0000
C01318=93.763,15.824,72.217,-177.0804,0.7487,0.0000
C01319=89.208,14.463,69.859,176.3869,-1.3548,0.0000
C01320=86.634,12.189,68.173,163.8300,-26.6085,0.0000
C01321=86.115,7.803,67.507,179.0232,-38.3726,0.0000
C01322=86.321,3.713,67.479,-177.7292,-38.8069,0.0000
C01323=86.399,0.000,67.498,-179.9997,-38.8306,0.0000
C01324=86.321,-3.713,67.479,177.7289,-38.8070,0.0000
C01325=86.115,-7.803,67.507,-179.0206,-38.3721,0.0000
C01326=86.634,-12.189,68.173,-163.8302,-26.6088,0.0000
C01327=89.208,-14.463,69.859,-176.3869,-1.3548,0.0000
C01328=93.763,-15.824,72.217,177.0804,0.7487,0.0000
C01329=99.916,-17.059,74.682,174.0572,1.3285,0.0000
C01330=106.881,-18.380,76.596,172.2484,1.8117,0.0000
C01331=113.357,-20.040,77.551,172.7181,3.4631,0.0000
C01332=118.041,-24.163,78.056,177.3136,4.1568,0.0000
C01333=120.177,-30.282,78.469,179.7520,2.4638,0.0000
C01334=119.269,-37.200,78.887,-179.9547,0.1510,0.0000
C01335=116.883,-44.288,79.163,-179.9933,0.0179,0.0000
C01336=113.965,-51.332,79.163,-179.9921,0.0174,0.0000
C01337=110.641,-58.031,78.887,-179.9253,0.1388,0.0000
C01338=106.390,-63.566,78.469,-178.0821,1.5675,0.0000
C01339=100.553,-66.382,78.056,-175.1661,1.0434,0.0000
C01340=94.325,-65.985,77.551,-172.4159,-2.7232,0.0000
C01341=88.573,-62.579,76.596,-173.2352,-4.2257,0.0000
C01342=82.714,-58.589,74.682,-174.8570,-3.2742,0.0000
C01343=77.490,-55.112,72.217,-177.4061,-1.5365,0.0000
C01344=73.307,-52.853,69.859,176.4881,1.5997,0.0000
C01345=69.878,-52.641,68.173,150.7837,-8.4855,0.0000
C01346=66.410,-55.375,67.507,150.2325,-28.7156,0.0000
C01347=63.664,-58.412,67.479,151.6030,-30.8249,0.0000
C01348=61.093,-61.093,67.498,150.3538,-29.6466,0.0000
C01349=58.413,-63.663,67.479,149.1749,-28.3969,0.0000
C01350=55.375,-66.410,67.507,151.2862,-29.7685,0.0000
C01351=52.641,-69.878,68.173,171.5141,-29.2165,0.0000
C01352=52.853,-73.307,69.859,-178.4003,-3.5119,0.0000
C01353=55.112,-77.490,72.217,178.4635,2.5939,0.0000
C01354=58.589,-82.714,74.682,176.7258,5.1430,0.0000
C01355=62.579,-88.573,76.596,175.7743,6.7648,0.0000
C01356=65.985,-94.325,77.551,177.2768,7.5841,0.0000
C01357=66.382,-100.553,78.056,-178.9566,4.8339,0.0000
C01358=63.566,-106.390,78.469,-178.4325,1.9179,0.0000
C01359=58.031,-110.641,78.887,-179.8612,0.0747,0.0000
C01360=51.332,-113.965,79.163,-179.9826,0.0079,0.0000
C01361=44.288,-116.883,79.163,-179.9821,0.0067,0.0000
C01362=37.200,-119.269,78.887,-179.8490,0.0453,0.0000
C01363=30.282,-120.177,78.469,-177.5362,-0.2480,0.0000
C01364=24.163,-118.041,78.056,-175.8432,-2.6864,0.0000
C01365=20.040,-113.357,77.551,-176.5369,-7.2819,0.0000
C01366=18.380,-106.881,76.596,-178.1883,-7.7516,0.0000
C01367=17.059,-99.916,74.682,-178.6715,-5.9428,0.0000
C01368=15.824,-93.763,72.217,-179.2513,-2.9196,0.0000
C01369=14.463,-89.208,69.859,178.6452,3.6131,0.0000
C01370=12.189,-86.634,68.173,153.3915,16.1700,0.0000
C01371=7.803,-86.115,67.507,141.6274,0.9768,0.0000
C01372=3.713,-86.321,67.479,141.1931,-2.2708,0.0000
C01373=0.000,-86.399,67.498,141.1694,-0.0003,0.0000
C01374=0.000,-86.399,67.498,141.1694,-0.0003,0.0000
C01375=-3.713,-86.321,67.479,141.1930,2.2711,0.0000
C01376=-7.803,-86.115,67.507,141.6279,-0.9794,0.0000
C01377=-12.189,-86.634,68.173,153.3912,-16.1698,0.0000
C01378=-14.463,-89.208,69.859,178.6452,-3.6131,0.0000
C01379=-15.824,-93.763,72.217,-179.2513,2.9196,0.0000
C01380=-17.059,-99.916,74.682,-178.6715,5.9428,0.0000
C01381=-18.380,-106.881,76.596,-178.1883,7.7516,0.0000
C01382=-20.040,-113.357,77.551,-176.5369,7.2819,0.0000
C01383=-24.163,-118.041,78.056,-175.8432,2.6864,0.0000
C01384=-30.282,-120.177,78.469,-177.5362,0.2480,0.0000
C01385=-37.200,-119.269,78.887,-179.8490,-0.0453,0.0000
C01386=-44.288,-116.883,79.163,-179.9821,-0.0067,0.0000
C01387=-51.332,-113.965,79.163,-179.9826,-0.0079,0.0000
C01388=-58.031,-110.641,78.887,-179.8612,-0.0747,0.0000
C01389=-63.566,-106.390,78.469,-178.4325,-1.9179,0.0000
C01390=-66.382,-100.553,78.056,-178.9566,-4.8339,0.0000
C01391=-65.985,-94.325,77.551,177.2768,-7.5841,0.0000
C01392=-62.579,-88.573,76.596,175.7743,-6.7648,0.0000
C01393=-58.589,-82.714,74.682,176.7258,-5.1430,0.0000
C01394=-55.112,-77.490,72.217,178.4635,-2.5939,0.0000
C01395=-52.853,-73.307,69.859,-178.4003,3.5119,0.0000
C01396=-52.641,-69.878,68.173,171.5145,29.2163,0.0000
C01397=-55.375,-66.410,67.507,151.2844,29.7675,0.0000
C01398=-58.412,-63.664,67.479,149.1751,28.3970,0.0000
C01399=-61.093,-61.093,67.498,150.3534,29.6462,0.0000
C01400=-63.663,-58.413,67.479,151.6031,30.8251,0.0000
C01401=-66.410,-55.375,67.507,150.2315,28.7138,0.0000
C01402=-69.878,-52.641,68.173,150.7835,8.4859,0.0000
C01403=-73.307,-52.853,69.859,176.4881,-1.5997,0.0000
C01404=-77.490,-55.112,72.217,-177.4061,1.5365,0.0000
C01405=-82.714,-58.589,74.682,-174.8570,3.2742,0.0000
C01406=-88.573,-62.579,76.596,-173.2352,4.2257,0.0000
C01407=-94.325,-65.985,77.551,-172.4159,2.7232,0.0000
C01408=-100.553,-66.382,78.056,-175.1661,-1.0434,0.0000
C01409=-106.390,-63.566,78.469,-178.0821,-1.5675,0.0000
C01410=-110.641,-58.031,78.887,-179.9253,-0.1388,0.0000
C01411=-113.965,-51.332,79.163,-179.9921,-0.0174,0.0000
C01412=-116.883,-44.288,79.163,-179.9933,-0.0179,0.0000
C01413=-119.269,-37.200,78.887,-179.9547,-0.1510,0.0000
C01414=-120.177,-30.282,78.469,179.7520,-2.4638,0.0000
C01415=-118.041,-24.163,78.056,177.3136,-4.1568,0.0000
C01416=-113.357,-20.040,77.551,172.7181,-3.4631,0.0000
C01417=-106.881,-18.380,76.596,172.2484,-1.8117,0.0000
C01418=-99.916,-17.059,74.682,174.0572,-1.3285,0.0000
C01419=-93.763,-15.824,72.217,177.0804,-0.7487,0.0000
C01420=-89.208,-14.463,69.859,-176.3869,1.3548,0.0000
C01421=-86.634,-12.189,68.173,-163.8300,26.6085,0.0000
C01422=-86.115,-7.803,67.507,-179.0232,38.3726,0.0000
C01423=-86.321,-3.713,67.479,177.7292,38.8069,0.0000
C01424=-86.399,0.000,67.498,179.9997,38.8306,0.0000
C01425=-86.321,3.713,67.479,-177.7289,38.8070,0.0000
C01426=-86.115,7.803,67.507,179.0206,38.3721,0.0000
C01427=-86.634,12.189,68.173,163.8302,26.6088,0.0000
C01428=-89.208,14.463,69.859,176.3869,1.3548,0.0000
C01429=-93.763,15.824,72.217,-177.0804,-0.7487,0.0000
C01430=-99.916,17.059,74.682,-174.0572,-1.3285,0.0000
C01431=-106.881,18.380,76.596,-172.2484,-1.8117,0.0000
C01432=-113.357,20.040,77.551,-172.7181,-3.4631,0.0000
C01433=-118.041,24.163,78.056,-177.3136,-4.1568,0.0000
C01434=-120.177,30.282,78.469,-179.7520,-2.4638,0.0000
C01435=-119.269,37.200,78.887,179.9547,-0.1510,0.0000
C01436=-116.883,44.288,79.163,179.9933,-0.0179,0.0000
C01437=-113.965,51.332,79.163,179.9921,-0.0174,0.0000
C01438=-110.641,58.031,78.887,179.9253,-0.1388,0.0000
C01439=-106.390,63.566,78.469,178.0821,-1.5675,0.0000
C01440=-100.553,66.382,78.056,175.1661,-1.0434,0.0000
C01441=-94.325,65.985,77.551,172.4159,2.7232,0.0000
C01442=-88.573,62.579,76.596,173.2352,4.2257,0.0000
C01443=-82.714,58.589,74.682,174.8570,3.2742,0.0000
C01444=-77.490,55.112,72.217,177.4061,1.5365,0.0000
C01445=-73.307,52.853,69.859,-176.4881,-1.5997,0.0000
C01446=-69.878,52.641,68.173,-150.7837,8.4855,0.0000
C01447=-66.410,55.375,67.507,-150.2325,28.7156,0.0000
C01448=-63.664,58.412,67.479,-151.6030,30.8249,0.0000
C01449=-61.093,61.093,67.498,-150.3538,29.6466,0.0000
C01450=-58.413,63.663,67.479,-149.1749,28.3969,0.0000
C01451=-55.375,66.410,67.507,-151.2862,29.7685,0.0000
C01452=-52.641,69.878,68.173,-171.5141,29.2165,0.0000
C01453=-52.853,73.307,69.859,178.4003,3.5119,0.0000
C01454=-55.112,77.490,72.217,-178.4635,-2.5939,0.0000
C01455=-58.589,82.714,74.682,-176.7258,-5.1430,0.0000
C01456=-62.579,88.573,76.596,-175.7743,-6.7648,0.0000
C01457=-65.985,94.325,77.551,-177.2768,-7.5841,0.0000
C01458=-66.382,100.553,78.056,178.9566,-4.8339,0.0000
C01459=-63.566,106.390,78.469,178.4325,-1.9179,0.0000
C01460=-58.031,110.641,78.887,179.8612,-0.0747,0.0000
C01461=-51.332,113.965,79.163,179.9826,-0.0079,0.0000
C01462=-44.288,116.883,79.163,179.9821,-0.0067,0.0000
C01463=-37.200,119.269,78.887,179.8490,-0.0453,0.0000
C01464=-30.282,120.177,78.469,177.5362,0.2480,0.0000
C01465=-24.163,118.041,78.056,175.8432,2.6864,0.0000
C01466=-20.040,113.357,77.551,176.5369,7.2819,0.0000
C01467=-18.380,106.881,76.596,178.1883,7.7516,0.0000
C01468=-17.059,99.916,74.682,178.6715,5.9428,0.0000
C01469=-15.824,93.763,72.217,179.2513,2.9196,0.0000
C01470=-14.463,89.208,69.859,-178.6452,-3.6131,0.0000
C01471=-12.189,86.634,68.173,-153.3912,-16.1698,0.0000
C01472=-7.803,86.115,67.507,-141.6279,-0.9794,0.0000
C01473=-3.713,86.321,67.479,-141.1930,2.2711,0.0000
C01474=0.000,86.399,67.498,-141.1694,-0.0003,0.0000
C01475=0.000,85.023,69.214,-141.4044,-0.0004,0.0000
C01476=3.588,84.949,69.194,-141.4273,-2.2241,0.0000
C01477=7.591,84.756,69.224,-141.8999,1.2653,0.0000
C01478=11.930,85.321,69.919,-154.4293,16.3224,0.0000
C01479=14.147,88.015,71.680,-178.9925,2.8637,0.0000
C01480=15.463,92.759,74.141,179.2095,-3.2389,0.0000
C01481=16.670,99.156,76.709,178.7065,-6.0491,0.0000
C01482=17.967,106.389,78.701,178.2758,-7.7577,0.0000
C01483=19.594,113.114,79.691,176.6650,-7.3174,0.0000
C01484=23.745,117.991,80.215,175.8678,-2.7559,0.0000
C01485=29.952,120.237,80.643,177.5407,-0.2660,0.0000
C01486=36.992,119.338,81.076,179.8480,0.0455,0.0000
C01487=44.218,116.910,81.361,179.9821,0.0067,0.0000
C01488=51.401,113.935,81.361,179.9826,0.0079,0.0000
C01489=58.227,110.542,81.076,179.8603,0.0753,0.0000
C01490=63.842,106.199,80.643,178.4484,1.9275,0.0000
C01491=66.642,100.222,80.215,179.0233,4.8654,0.0000
C01492=66.129,93.838,79.691,-177.1607,7.5199,0.0000
C01493=62.524,87.933,78.701,-175.7083,6.7080,0.0000
C01494=58.326,81.902,76.709,-176.6254,5.1939,0.0000
C01495=54.657,76.524,74.141,-178.2668,2.8494,0.0000
C01496=52.233,72.239,71.680,178.6861,-2.7370,0.0000
C01497=51.896,68.767,69.919,-172.5214,-28.6088,0.0000
C01498=54.564,65.299,69.224,-151.6831,-29.6858,0.0000
C01499=57.531,62.605,69.194,-149.4005,-28.2119,0.0000
C01500=60.120,60.120,69.214,-150.5600,-29.4396,0.0000
C01501=62.605,57.532,69.194,-151.7883,-30.5998,0.0000
C01502=65.300,54.563,69.224,-150.3131,-28.3150,0.0000
C01503=68.767,51.896,69.919,-151.3911,-7.4789,0.0000
C01504=72.239,52.233,71.680,-177.2630,1.3139,0.0000
C01505=76.524,54.657,74.141,177.1506,-1.7332,0.0000
C01506=81.902,58.326,76.709,174.8061,-3.3746,0.0000
C01507=87.933,62.524,78.701,173.2920,-4.2917,0.0000
C01508=93.838,66.129,79.691,172.4801,-2.8393,0.0000
C01509=100.222,66.642,80.215,175.1346,0.9767,0.0000
C01510=106.199,63.842,80.643,178.0725,1.5516,0.0000
C01511=110.542,58.227,81.076,179.9247,0.1397,0.0000
C01512=113.935,51.401,81.361,179.9921,0.0174,0.0000
C01513=116.910,44.218,81.361,179.9933,0.0179,0.0000
C01514=119.338,36.992,81.076,179.9545,0.1520,0.0000
C01515=120.237,29.952,80.643,-179.7340,2.4593,0.0000
C01516=117.991,23.745,80.215,-177.2441,4.1322,0.0000
C01517=113.114,19.594,79.691,-172.6826,3.3350,0.0000
C01518=106.389,17.967,78.701,-172.2423,1.7242,0.0000
C01519=99.156,16.670,76.709,-173.9509,1.2935,0.0000
C01520=92.759,15.463,74.141,-176.7611,0.7905,0.0000
C01521=88.015,14.147,71.680,177.1363,-1.0075,0.0000
C01522=85.321,11.930,69.919,163.6776,-25.5707,0.0000
C01523=84.756,7.591,69.224,178.7347,-38.1001,0.0000
C01524=84.949,3.588,69.194,-177.7759,-38.5727,0.0000
C01525=85.023,0.000,69.214,-179.9996,-38.5956,0.0000
C01526=84.949,-3.587,69.194,177.7755,-38.5728,0.0000
C01527=84.756,-7.592,69.224,-178.7320,-38.0996,0.0000
C01528=85.322,-11.930,69.919,-163.6777,-25.5710,0.0000
C01529=88.015,-14.147,71.680,-177.1363,-1.0075,0.0000
C01530=92.759,-15.463,74.141,176.7611,0.7905,0.0000
C01531=99.156,-16.670,76.709,173.9509,1.2935,0.0000
C01532=106.389,-17.967,78.701,172.2423,1.7242,0.0000
C01533=113.114,-19.594,79.691,172.6826,3.3350,0.0000
C01534=117.991,-23.745,80.215,177.2441,4.1322,0.0000
C01535=120.237,-29.952,80.643,179.7340,2.4593,0.0000
C01536=119.338,-36.992,81.076,-179.9545,0.1520,0.0000
C01537=116.910,-44.218,81.361,-179.9933,0.0179,0.0000
C01538=113.935,-51.401,81.361,-179.9921,0.0174,0.0000
C01539=110.542,-58.227,81.076,-179.9247,0.1397,0.0000
C01540=106.199,-63.842,80.643,-178.0725,1.5516,0.0000
C01541=100.222,-66.642,80.215,-175.1346,0.9767,0.0000
C01542=93.838,-66.129,79.691,-172.4801,-2.8393,0.0000
C01543=87.933,-62.524,78.701,-173.2920,-4.2917,0.0000
C01544=81.902,-58.326,76.709,-174.8061,-3.3746,0.0000
C01545=76.524,-54.657,74.141,-177.1506,-1.7332,0.0000
C01546=72.239,-52.233,71.680,177.2630,1.3139,0.0000
C01547=68.767,-51.896,69.919,151.3912,-7.4786,0.0000
C01548=65.299,-54.564,69.224,150.3142,-28.3169,0.0000
C01549=62.605,-57.531,69.194,151.7881,-30.5995,0.0000
C01550=60.120,-60.120,69.214,150.5604,-29.4400,0.0000
C01551=57.532,-62.605,69.194,149.4002,-28.2117,0.0000
C01552=54.563,-65.300,69.224,151.6850,-29.6869,0.0000
C01553=51.896,-68.767,69.919,172.5211,-28.6089,0.0000
C01554=52.233,-72.239,71.680,-178.6861,-2.7370,0.0000
C01555=54.657,-76.524,74.141,178.2668,2.8494,0.0000
C01556=58.326,-81.902,76.709,176.6254,5.1939,0.0000
C01557=62.524,-87.933,78.701,175.7083,6.7080,0.0000
C01558=66.129,-93.838,79.691,177.1607,7.5199,0.0000
C01559=66.642,-100.222,80.215,-179.0233,4.8654,0.0000
C01560=63.842,-106.199,80.643,-178.4484,1.9275,0.0000
C01561=58.227,-110.542,81.076,-179.8603,0.0753,0.0000
C01562=51.401,-113.935,81.361,-179.9826,0.0079,0.0000
C01563=44.218,-116.910,81.361,-179.9821,0.0067,0.0000
C01564=36.992,-119.338,81.076,-179.8480,0.0455,0.0000
C01565=29.952,-120.237,80.643,-177.5407,-0.2660,0.0000
C01566=23.745,-117.991,80.215,-175.8678,-2.7559,0.0000
C01567=19.594,-113.114,79.691,-176.6650,-7.3174,0.0000
C01568=17.967,-106.389,78.701,-178.2758,-7.7577,0.0000
C01569=16.670,-99.156,76.709,-178.7065,-6.0491,0.0000
C01570=15.463,-92.759,74.141,-179.2095,-3.2389,0.0000
C01571=14.147,-88.015,71.680,178.9925,2.8637,0.0000
C01572=11.930,-85.321,69.919,154.4293,16.3224,0.0000
C01573=7.591,-84.756,69.224,141.8999,1.2653,0.0000
C01574=3.588,-84.949,69.194,141.4273,-2.2241,0.0000
C01575=0.000,-85.023,69.214,141.4044,-0.0004,0.0000
C01576=0.000,-85.023,69.214,141.4044,-0.0004,0.0000
C01577=-3.587,-84.949,69.194,141.4272,2.2245,0.0000
C01578=-7.592,-84.756,69.224,141.9004,-1.2680,0.0000
C01579=-11.930,-85.322,69.919,154.4290,-16.3223,0.0000
C01580=-14.147,-88.015,71.680,178.9925,-2.8637,0.0000
C01581=-15.463,-92.759,74.141,-179.2095,3.2389,0.0000
C01582=-16.670,-99.156,76.709,-178.7065,6.0491,0.0000
C01583=-17.967,-106.389,78.701,-178.2758,7.7577,0.0000
C01584=-19.594,-113.114,79.691,-176.6650,7.3174,0.0000
C01585=-23.745,-117.991,80.215,-175.8678,2.7559,0.0000
C01586=-29.952,-120.237,80.643,-177.5407,0.2660,0.0000
C01587=-36.992,-119.338,81.076,-179.8480,-0.0455,0.0000
C01588=-44.218,-116.910,81.361,-179.9821,-0.0067,0.0000
C01589=-51.401,-113.935,81.361,-179.9826,-0.0079,0.0000
C01590=-58.227,-110.542,81.076,-179.8603,-0.0753,0.0000
C01591=-63.842,-106.199,80.643,-178.4484,-1.9275,0.0000
C01592=-66.642,-100.222,80.215,-179.0233,-4.8654,0.0000
C01593=-66.129,-93.838,79.691,177.1607,-7.5199,0.0000
C01594=-62.524,-87.933,78.701,175.7083,-6.7080,0.0000
C01595=-58.326,-81.902,76.709,176.6254,-5.1939,0.0000
C01596=-54.657,-76.524,74.141,178.2668,-2.8494,0.0000
C01597=-52.233,-72.239,71.680,-178.6861,2.7370,0.0000
C01598=-51.896,-68.767,69.919,172.5214,28.6088,0.0000
C01599=-54.564,-65.299,69.224,151.6831,29.6858,0.0000
C01600=-57.531,-62.605,69.194,149.4005,28.2119,0.0000
C01601=-60.120,-60.120,69.214,150.5600,29.4396,0.0000
C01602=-62.605,-57.532,69.194,151.7883,30.5998,0.0000
C01603=-65.300,-54.563,69.224,150.3131,28.3150,0.0000
C01604=-68.767,-51.896,69.919,151.3911,7.4789,0.0000
C01605=-72.239,-52.233,71.680,177.2630,-1.3139,0.0000
C01606=-76.524,-54.657,74.141,-177.1506,1.7332,0.0000
C01607=-81.902,-58.326,76.709,-174.8061,3.3746,0.0000
C01608=-87.933,-62.524,78.701,-173.2920,4.2917,0.0000
C01609=-93.838,-66.129,79.691,-172.4801,2.8393,0.0000
C01610=-100.222,-66.642,80.215,-175.1346,-0.9767,0.0000
C01611=-106.199,-63.842,80.643,-178.0725,-1.5516,0.0000
C01612=-110.542,-58.227,81.076,-179.9247,-0.1397,0.0000
C01613=-113.935,-51.401,81.361,-179.9921,-0.0174,0.0000
C01614=-116.910,-44.218,81.361,-179.9933,-0.0179,0.0000
C01615=-119.338,-36.992,81.076,-179.9545,-0.1520,0.0000
C01616=-120.237,-29.952,80.643,179.7340,-2.4593,0.0000
C01617=-117.991,-23.745,80.215,177.2441,-4.1322,0.0000
C01618=-113.114,-19.594,79.691,172.6826,-3.3350,0.0000
C01619=-106.389,-17.967,78.701,172.2423,-1.7242,0.0000
C01620=-99.156,-16.670,76.709,173.9509,-1.2935,0.0000
C01621=-92.759,-15.463,74.141,176.7611,-0.7905,0.0000
C01622=-88.015,-14.147,71.680,-177.1363,1.0075,0.0000
C01623=-85.321,-11.930,69.919,-163.6776,25.5707,0.0000
C01624=-84.756,-7.591,69.224,-178.7347,38.1001,0.0000
C01625=-84.949,-3.588,69.194,177.7759,38.5727,0.0000
C01626=-85.023,0.000,69.214,179.9996,38.5956,0.0000
C01627=-84.949,3.587,69.194,-177.7755,38.5728,0.0000
C01628=-84.756,7.592,69.224,178.7320,38.0996,0.0000
C01629=-85.322,11.930,69.919,163.6777,25.5710,0.0000
C01630=-88.015,14.147,71.680,177.1363,1.0075,0.0000
C01631=-92.759,15.463,74.141,-176.7611,-0.7905,0.0000
C01632=-99.156,16.670,76.709,-173.9509,-1.2935,0.0000
C01633=-106.389,17.967,78.701,-172.2423,-1.7242,0.0000
C01634=-113.114,19.594,79.691,-172.6826,-3.3350,0.0000
C01635=-117.991,23.745,80.215,-177.2441,-4.1322,0.0000
C01636=-120.237,29.952,80.643,-179.7340,-2.4593,0.0000
C01637=-119.338,36.992,81.076,179.9545,-0.1520,0.0000
C01638=-116.910,44.218,81.361,179.9933,-0.0179,0.0000
C01639=-113.935,51.401,81.361,179.9921,-0.0174,0.0000
C01640=-110.542,58.227,81.076,179.9247,-0.1397,0.0000
C01641=-106.199,63.842,80.643,178.0725,-1.5516,0.0000
C01642=-100.222,66.642,80.215,175.1346,-0.9767,0.0000
C01643=-93.838,66.129,79.691,172.4801,2.8393,0.0000
C01644=-87.933,62.524,78.701,173.2920,4.2917,0.0000
C01645=-81.902,58.326,76.709,174.8061,3.3746,0.0000
C01646=-76.524,54.657,74.141,177.1506,1.7332,0.0000
C01647=-72.239,52.233,71.680,-177.2630,-1.3139,0.0000
C01648=-68.767,51.896,69.919,-151.3912,7.4786,0.0000
C01649=-65.299,54.564,69.224,-150.3142,28.3169,0.0000
C01650=-62.605,57.531,69.194,-151.7881,30.5995,0.0000
C01651=-60.120,60.120,69.214,-150.5604,29.4400,0.0000
C01652=-57.532,62.605,69.194,-149.4002,28.2117,0.0000
C01653=-54.563,65.300,69.224,-151.6850,29.6869,0.0000
C01654=-51.896,68.767,69.919,-172.5211,28.6089,0.0000
C01655=-52.233,72.239,71.680,178.6861,2.7370,0.0000
C01656=-54.657,76.524,74.141,-178.2668,-2.8494,0.0000
C01657=-58.326,81.902,76.709,-176.6254,-5.1939,0.0000
C01658=-62.524,87.933,78.701,-175.7083,-6.7080,0.0000
C01659=-66.129,93.838,79.691,-177.1607,-7.5199,0.0000
C01660=-66.642,100.222,80.215,179.0233,-4.8654,0.0000
C01661=-63.842,106.199,80.643,178.4484,-1.9275,0.0000
C01662=-58.227,110.542,81.076,179.8603,-0.0753,0.0000
C01663=-51.401,113.935,81.361,179.9826,-0.0079,0.0000
C01664=-44.218,116.910,81.361,179.9821,-0.0067,0.0000
C01665=-36.992,119.338,81.076,179.8480,-0.0455,0.0000
C01666=-29.952,120.237,80.643,177.5407,0.2660,0.0000
C01667=-23.745,117.991,80.215,175.8678,2.7559,0.0000
C01668=-19.594,113.114,79.691,176.6650,7.3174,0.0000
C01669=-17.967,106.389,78.701,178.2758,7.7577,0.0000
C01670=-16.670,99.156,76.709,178.7065,6.0491,0.0000
C01671=-15.463,92.759,74.141,179.2095,3.2389,0.0000
C01672=-14.147,88.015,71.680,-178.9925,-2.8637,0.0000
C01673=-11.930,85.322,69.919,-154.4290,-16.3223,0.0000
C01674=-7.592,84.756,69.224,-141.9004,-1.2680,0.0000
C01675=-3.587,84.949,69.194,-141.4272,2.2245,0.0000
C01676=0.000,85.023,69.214,-141.4044,-0.0004,0.0000
C01677=0.000,83.655,70.937,-141.6907,-0.0005,0.0000
C01678=3.463,83.586,70.916,-141.7127,-2.1723,0.0000
C01679=7.381,83.405,70.947,-142.2267,1.5514,0.0000
C01680=11.673,84.017,71.672,-155.5055,16.3902,0.0000
C01681=13.833,86.832,73.509,-179.2852,2.1623,0.0000
C01682=15.106,91.768,76.072,179.1825,-3.5126,0.0000
C01683=16.288,98.410,78.743,178.7471,-6.1136,0.0000
C01684=17.564,105.909,80.809,178.3653,-7.7182,0.0000
C01685=19.159,112.877,81.835,176.8028,-7.3030,0.0000
C01686=23.337,117.942,82.377,175.9177,-2.8029,0.0000
C01687=29.630,120.296,82.819,177.5597,-0.2812,0.0000
C01688=36.790,119.404,83.265,179.8481,0.0453,0.0000
C01689=44.150,116.936,83.560,179.9822,0.0067,0.0000
C01690=51.468,113.905,83.560,179.9827,0.0079,0.0000
C01691=58.417,110.446,83.265,179.8605,0.0754,0.0000
C01692=64.110,106.014,82.819,178.4726,1.9247,0.0000
C01693=66.895,99.899,82.377,179.0921,4.8634,0.0000
C01694=66.269,93.364,81.835,-177.0735,7.4135,0.0000
C01695=62.469,87.308,80.809,-175.6736,6.6174,0.0000
C01696=58.069,81.104,78.743,-176.5509,5.2111,0.0000
C01697=54.208,75.571,76.072,-178.0919,3.0621,0.0000
C01698=51.618,71.181,73.509,178.9759,-2.0343,0.0000
C01699=51.155,67.663,71.672,-173.4859,-27.9301,0.0000
C01700=53.757,64.195,70.947,-152.1297,-29.5581,0.0000
C01701=56.656,61.552,70.916,-149.6721,-27.9845,0.0000
C01702=59.153,59.153,70.937,-150.8109,-29.1886,0.0000
C01703=61.552,56.656,70.916,-152.0157,-30.3282,0.0000
C01704=64.195,53.757,70.948,-150.4409,-27.8684,0.0000
C01705=67.663,51.155,71.672,-152.0698,-6.5143,0.0000
C01706=71.181,51.618,73.509,-177.9657,1.0241,0.0000
C01707=75.571,54.208,76.072,176.9379,-1.9081,0.0000
C01708=81.104,58.069,78.743,174.7889,-3.4491,0.0000
C01709=87.308,62.469,80.809,173.3826,-4.3264,0.0000
C01710=93.364,66.269,81.835,172.5865,-2.9265,0.0000
C01711=99.899,66.895,82.377,175.1366,0.9079,0.0000
C01712=106.014,64.110,82.819,178.0753,1.5274,0.0000
C01713=110.446,58.417,83.265,179.9246,0.1395,0.0000
C01714=113.905,51.468,83.560,179.9921,0.0173,0.0000
C01715=116.936,44.150,83.560,179.9933,0.0178,0.0000
C01716=119.404,36.790,83.265,179.9547,0.1519,0.0000
C01717=120.296,29.630,82.819,-179.7188,2.4403,0.0000
C01718=117.942,23.337,82.377,-177.1971,4.0823,0.0000
C01719=112.877,19.159,81.835,-172.6970,3.1972,0.0000
C01720=105.909,17.564,80.809,-172.2818,1.6347,0.0000
C01721=98.410,16.288,78.743,-173.8864,1.2529,0.0000
C01722=91.768,15.106,76.072,-176.4874,0.8175,0.0000
C01723=86.832,13.833,73.509,177.8377,-0.7148,0.0000
C01724=84.017,11.673,71.672,163.6098,-24.4945,0.0000
C01725=83.405,7.381,70.947,178.4486,-37.7733,0.0000
C01726=83.586,3.463,70.916,-177.8277,-38.2873,0.0000
C01727=83.655,0.000,70.937,-179.9995,-38.3093,0.0000
C01728=83.586,-3.462,70.916,177.8272,-38.2873,0.0000
C01729=83.405,-7.381,70.948,-178.4459,-37.7728,0.0000
C01730=84.017,-11.673,71.672,-163.6099,-24.4947,0.0000
C01731=86.832,-13.833,73.509,-177.8377,-0.7148,0.0000
C01732=91.768,-15.106,76.072,176.4874,0.8175,0.0000
C01733=98.410,-16.288,78.743,173.8864,1.2529,0.0000
C01734=105.909,-17.564,80.809,172.2818,1.6347,0.0000
C01735=112.877,-19.159,81.835,172.6970,3.1972,0.0000
C01736=117.942,-23.337,82.377,177.1971,4.0823,0.0000
C01737=120.296,-29.630,82.819,179.7188,2.4403,0.0000
C01738=119.404,-36.790,83.265,-179.9547,0.1519,0.0000
C01739=116.936,-44.150,83.560,-179.9933,0.0178,0.0000
C01740=113.905,-51.468,83.560,-179.9921,0.0173,0.0000
C01741=110.446,-58.417,83.265,-179.9246,0.1395,0.0000
C01742=106.014,-64.110,82.819,-178.0753,1.5274,0.0000
C01743=99.899,-66.895,82.377,-175.1366,0.9079,0.0000
C01744=93.364,-66.269,81.835,-172.5865,-2.9265,0.0000
C01745=87.308,-62.469,80.809,-173.3826,-4.3264,0.0000
C01746=81.104,-58.069,78.743,-174.7889,-3.4491,0.0000
C01747=75.571,-54.208,76.072,-176.9379,-1.9081,0.0000
C01748=71.181,-51.618,73.509,177.9657,1.0241,0.0000
C01749=67.663,-51.155,71.672,152.0699,-6.5141,0.0000
C01750=64.195,-53.757,70.947,150.4419,-27.8703,0.0000
C01751=61.552,-56.656,70.916,152.0155,-30.3279,0.0000
C01752=59.153,-59.153,70.937,150.8114,-29.1891,0.0000
C01753=56.656,-61.552,70.916,149.6718,-27.9843,0.0000
C01754=53.757,-64.195,70.948,152.1316,-29.5591,0.0000
C01755=51.155,-67.663,71.672,173.4857,-27.9302,0.0000
C01756=51.618,-71.181,73.509,-178.9759,-2.0343,0.0000
C01757=54.208,-75.571,76.072,178.0919,3.0621,0.0000
C01758=58.069,-81.104,78.743,176.5509,5.2111,0.0000
C01759=62.469,-87.308,80.809,175.6736,6.6174,0.0000
C01760=66.269,-93.364,81.835,177.0735,7.4135,0.0000
C01761=66.895,-99.899,82.377,-179.0921,4.8634,0.0000
C01762=64.110,-106.014,82.819,-178.4726,1.9247,0.0000
C01763=58.417,-110.446,83.265,-179.8605,0.0754,0.0000
C01764=51.468,-113.905,83.560,-179.9827,0.0079,0.0000
C01765=44.150,-116.936,83.560,-179.9822,0.0067,0.0000
C01766=36.790,-119.404,83.265,-179.8481,0.0453,0.0000
C01767=29.630,-120.296,82.819,-177.5597,-0.2812,0.0000
C01768=23.337,-117.942,82.377,-175.9177,-2.8029,0.0000
C01769=19.159,-112.877,81.835,-176.8028,-7.3030,0.0000
C01770=17.564,-105.909,80.809,-178.3653,-7.7182,0.0000
C01771=16.288,-98.410,78.743,-178.7471,-6.1136,0.0000
C01772=15.106,-91.768,76.072,-179.1825,-3.5126,0.0000
C01773=13.833,-86.832,73.509,179.2852,2.1623,0.0000
C01774=11.673,-84.017,71.672,155.5055,16.3902,0.0000
C01775=7.381,-83.405,70.947,142.2267,1.5514,0.0000
C01776=3.463,-83.586,70.916,141.7127,-2.1723,0.0000
C01777=0.000,-83.655,70.937,141.6907,-0.0005,0.0000
C01778=0.000,-83.655,70.937,141.6907,-0.0005,0.0000
C01779=-3.462,-83.586,70.916,141.7127,2.1728,0.0000
C01780=-7.381,-83.405,70.948,142.2272,-1.5541,0.0000
C01781=-11.673,-84.017,71.672,155.5053,-16.3901,0.0000
C01782=-13.833,-86.832,73.509,179.2852,-2.1623,0.0000
C01783=-15.106,-91.768,76.072,-179.1825,3.5126,0.0000
C01784=-16.288,-98.410,78.743,-178.7471,6.1136,0.0000
C01785=-17.564,-105.909,80.809,-178.3653,7.7182,0.0000
C01786=-19.159,-112.877,81.835,-176.8028,7.3030,0.0000
C01787=-23.337,-117.942,82.377,-175.9177,2.8029,0.0000
C01788=-29.630,-120.296,82.819,-177.5597,0.2812,0.0000
C01789=-36.790,-119.404,83.265,-179.8481,-0.0453,0.0000
C01790=-44.150,-116.936,83.560,-179.9822,-0.0067,0.0000
C01791=-51.468,-113.905,83.560,-179.9827,-0.0079,0.0000
C01792=-58.417,-110.446,83.265,-179.8605,-0.0754,0.0000
C01793=-64.110,-106.014,82.819,-178.4726,-1.9247,0.0000
C01794=-66.895,-99.899,82.377,-179.0921,-4.8634,0.0000
C01795=-66.269,-93.364,81.835,177.0735,-7.4135,0.0000
C01796=-62.469,-87.308,80.809,175.6736,-6.6174,0.0000
C01797=-58.069,-81.104,78.743,176.5509,-5.2111,0.0000
C01798=-54.208,-75.571,76.072,178.0919,-3.0621,0.0000
C01799=-51.618,-71.181,73.509,-178.9759,2.0343,0.0000
C01800=-51.155,-67.663,71.672,173.4859,27.9301,0.0000
C01801=-53.757,-64.195,70.947,152.1297,29.5581,0.0000
C01802=-56.656,-61.552,70.916,149.6721,27.9845,0.0000
C01803=-59.153,-59.153,70.937,150.8109,29.1886,0.0000
C01804=-61.552,-56.656,70.916,152.0157,30.3282,0.0000
C01805=-64.195,-53.757,70.948,150.4409,27.8684,0.0000
C01806=-67.663,-51.155,71.672,152.0698,6.5143,0.0000
C01807=-71.181,-51.618,73.509,177.9657,-1.0241,0.0000
C01808=-75.571,-54.208,76.072,-176.9379,1.9081,0.0000
C01809=-81.104,-58.069,78.743,-174.7889,3.4491,0.0000
C01810=-87.308,-62.469,80.809,-173.3826,4.3264,0.0000
C01811=-93.364,-66.269,81.835,-172.5865,2.9265,0.0000
C01812=-99.899,-66.895,82.377,-175.1366,-0.9079,0.0000
C01813=-106.014,-64.110,82.819,-178.0753,-1.5274,0.0000
C01814=-110.446,-58.417,83.265,-179.9246,-0.1395,0.0000
C01815=-113.905,-51.468,83.560,-179.9921,-0.0173,0.0000
C01816=-116.936,-44.150,83.560,-179.9933,-0.0178,0.0000
C01817=-119.404,-36.790,83.265,-179.9547,-0.1519,0.0000
C01818=-120.296,-29.630,82.819,179.7188,-2.4403,0.0000
C01819=-117.942,-23.337,82.377,177.1971,-4.0823,0.0000
C01820=-112.877,-19.159,81.835,172.6970,-3.1972,0.0000
C01821=-105.909,-17.564,80.809,172.2818,-1.6347,0.0000
C01822=-98.410,-16.288,78.743,173.8864,-1.2529,0.0000
C01823=-91.768,-15.106,76.072,176.4874,-0.8175,0.0000
C01824=-86.832,-13.833,73.509,-177.8377,0.7148,0.0000
C01825=-84.017,-11.673,71.672,-163.6098,24.4945,0.0000
C01826=-83.405,-7.381,70.947,-178.4486,37.7733,0.0000
C01827=-83.586,-3.463,70.916,177.8277,38.2873,0.0000
C01828=-83.655,0.000,70.937,179.9995,38.3093,0.0000
C01829=-83.586,3.462,70.916,-177.8272,38.2873,0.0000
C01830=-83.405,7.381,70.948,178.4459,37.7728,0.0000
C01831=-84.017,11.673,71.672,163.6099,24.4947,0.0000
C01832=-86.832,13.833,73.509,177.8377,0.7148,0.0000
C01833=-91.768,15.106,76.072,-176.4874,-0.8175,0.0000
C01834=-98.410,16.288,78.743,-173.8864,-1.2529,0.0000
C01835=-105.909,17.564,80.809,-172.2818,-1.6347,0.0000
C01836=-112.877,19.159,81.835,-172.6970,-3.1972,0.0000
C01837=-117.942,23.337,82.377,-177.1971,-4.0823,0.0000
C01838=-120.296,29.630,82.819,-179.7188,-2.4403,0.0000
C01839=-119.404,36.790,83.265,179.9547,-0.1519,0.0000
C01840=-116.936,44.150,83.560,179.9933,-0.0178,0.0000
C01841=-113.905,51.468,83.560,179.9921,-0.0173,0.0000
C01842=-110.446,58.417,83.265,179.9246,-0.1395,0.0000
C01843=-106.014,64.110,82.819,178.0753,-1.5274,0.0000
C01844=-99.899,66.895,82.377,175.1366,-0.9079,0.0000
C01845=-93.364,66.269,81.835,172.5865,2.9265,0.0000
C01846=-87.308,62.469,80.809,173.3826,4.3264,0.0000
C01847=-81.104,58.069,78.743,174.7889,3.4491,0.0000
C01848=-75.571,54.208,76.072,176.9379,1.9081,0.0000
C01849=-71.181,51.618,73.509,-177.9657,-1.0241,0.0000
C01850=-67.663,51.155,71.672,-152.0699,6.5141,0.0000
C01851=-64.195,53.757,70.947,-150.4419,27.8703,0.0000
C01852=-61.552,56.656,70.916,-152.0155,30.3279,0.0000
C01853=-59.153,59.153,70.937,-150.8114,29.1891,0.0000
C01854=-56.656,61.552,70.916,-149.6718,27.9843,0.0000
C01855=-53.757,64.195,70.948,-152.1316,29.5591,0.0000
C01856=-51.155,67.663,71.672,-173.4857,27.9302,0.0000
C01857=-51.618,71.181,73.509,178.9759,2.0343,0.0000
C01858=-54.208,75.571,76.072,-178.0919,-3.0621,0.0000
C01859=-58.069,81.104,78.743,-176.5509,-5.2111,0.0000
C01860=-62.469,87.308,80.809,-175.6736,-6.6174,0.0000
